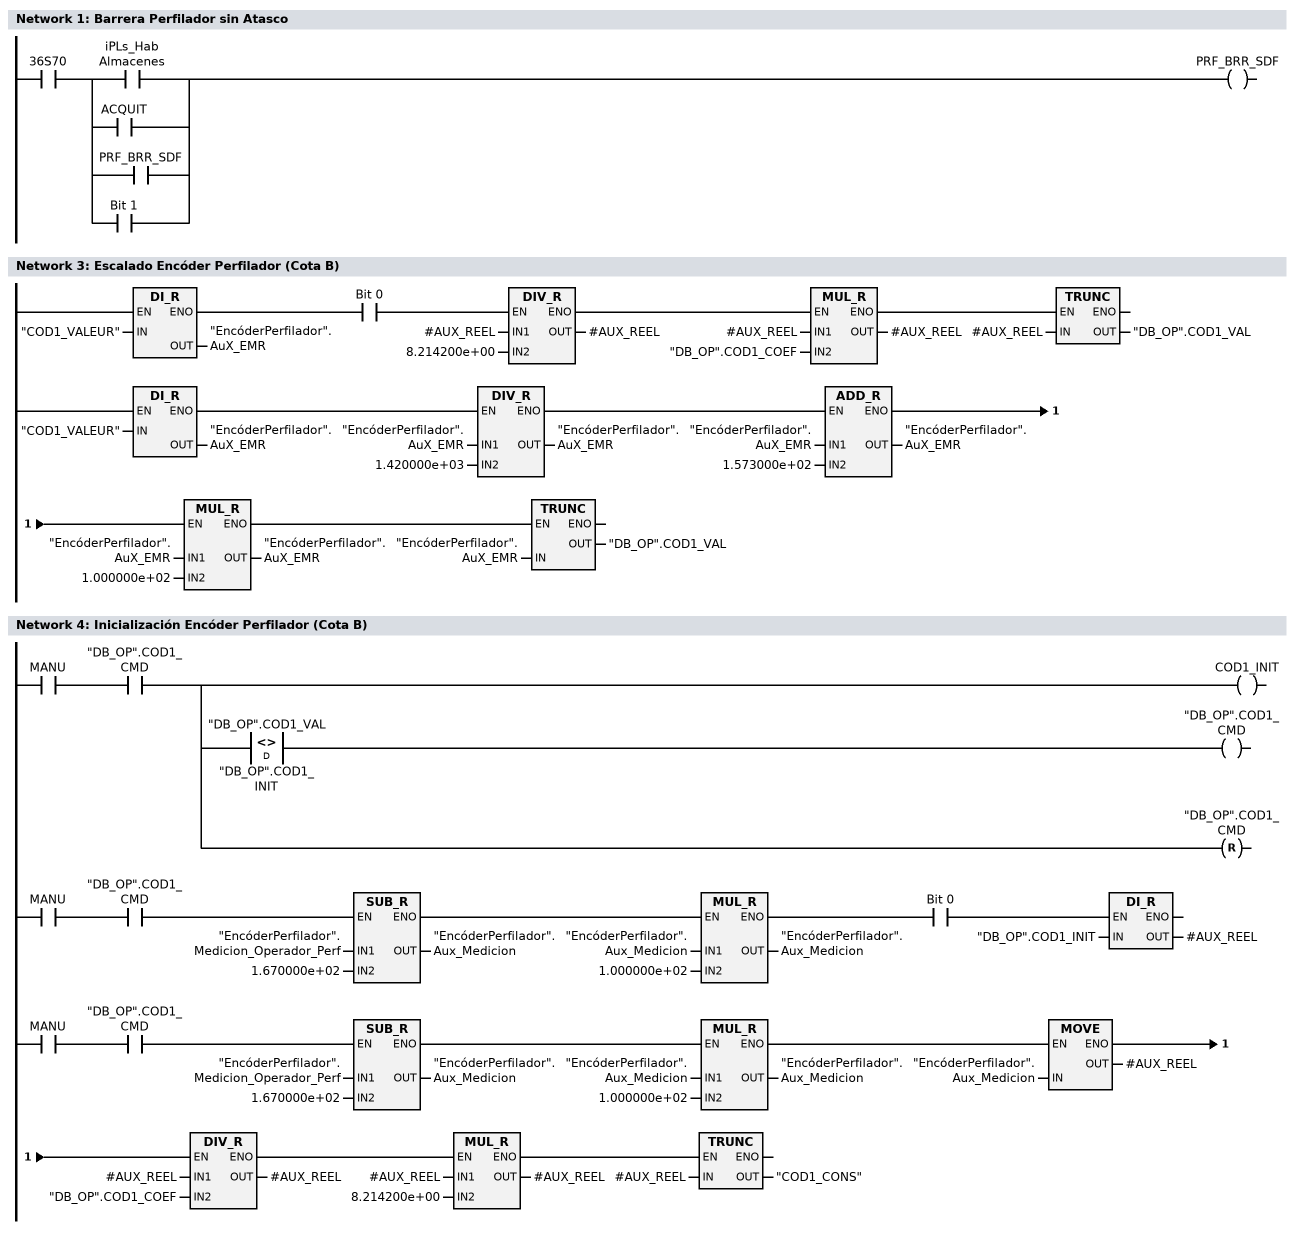
NETWORK
TITLE = Barrera Perfilador sin Atasco
      A     "36S70";
      A(;
      O     "iPLs_HabAlmacenes";
      O     "ACQUIT";
      O     "PRF_BRR_SDF";
      O     "Bit 1";
      );
      =     "PRF_BRR_SDF";
NETWORK
TITLE = Habilitación Infeed Perfiladora (CON/DES1)
      A     "Bit 1";
      A     "KMST";
      =     L 14.0;
      A(;
      A     L 14.0;
      AN    "PRF_SLM_LC";
      AN    "PRF_SLM_LS";
      AN    "PRF_SLM_SH";
      A     "PRF_SLM_BC";
      JNB   _001;
      L     1034;
      T     PQW 24;
      SET;
      SAVE;
      CLR;
_001: A     BR;
      );
      JNB   _002;
      L     1;
      T     PQW 28;
_002: NOP   0;
      A     L 14.0;
      A     "PRF_SLM_LC";
      AN    "PRF_SLM_BC";
      =     L 14.1;
      A(;
      A     L 14.1;
      AN    M 37.7;
      JNB   _003;
      L     1035;
      T     PQW 24;
      SET;
      SAVE;
      CLR;
_003: A     BR;
      );
      JNB   _004;
      L     1;
      T     PQW 28;
_004: NOP   0;
      A(;
      A     L 14.1;
      A     M 37.7;
      JNB   _005;
      L     0;
      T     PQW 24;
      SET;
      SAVE;
      CLR;
_005: A     BR;
      );
      JNB   _006;
      L     1;
      T     PQW 28;
_006: NOP   0;
NETWORK
TITLE = Escalado Encóder Perfilador (Cota B)
      L     "COD1_VALEUR";
      DTR;
      T     "EncóderPerfilador".AuX_EMR;
      SET;
      SAVE;
      CLR;
      A     BR;
      =     L 14.0;
      A(;
      A(;
      A     L 14.0;
      A     "Bit 0";
      JNB   _007;
      L     #AUX_REEL;
      L     8.214200e+00;
      /R;
      T     #AUX_REEL;
      AN    OV;
      SAVE;
      CLR;
_007: A     BR;
      );
      JNB   _008;
      L     #AUX_REEL;
      L     "DB_OP".COD1_COEF;
      *R;
      T     #AUX_REEL;
      AN    OV;
      SAVE;
      CLR;
_008: A     BR;
      );
      JNB   _009;
      L     #AUX_REEL;
      TRUNC;
      T     "DB_OP".COD1_VAL;
_009: NOP   0;
      A(;
      A(;
      A(;
      A     L 14.0;
      JNB   _00a;
      L     "EncóderPerfilador".AuX_EMR;
      L     1.420000e+03;
      /R;
      T     "EncóderPerfilador".AuX_EMR;
      AN    OV;
      SAVE;
      CLR;
_00a: A     BR;
      );
      JNB   _00b;
      L     "EncóderPerfilador".AuX_EMR;
      L     1.573000e+02;
      +R;
      T     "EncóderPerfilador".AuX_EMR;
      AN    OV;
      SAVE;
      CLR;
_00b: A     BR;
      );
      JNB   _00c;
      L     "EncóderPerfilador".AuX_EMR;
      L     1.000000e+02;
      *R;
      T     "EncóderPerfilador".AuX_EMR;
      AN    OV;
      SAVE;
      CLR;
_00c: A     BR;
      );
      JNB   _00d;
      L     "EncóderPerfilador".AuX_EMR;
      TRUNC;
      T     "DB_OP".COD1_VAL;
_00d: NOP   0;
NETWORK
TITLE = Inicialización Encóder Perfilador (Cota B)
      A     "MANU";
      A     "DB_OP".COD1_CMD;
      =     L 14.0;
      A(;
      A     L 14.0;
      JNB   _00e;
      L     "EncóderPerfilador".Medicion_Operador_Perf;
      L     1.670000e+02;
      -R;
      T     "EncóderPerfilador".Aux_Medicion;
      AN    OV;
      SAVE;
      CLR;
_00e: A     BR;
      );
      JNB   _00f;
      L     "EncóderPerfilador".Aux_Medicion;
      L     1.000000e+02;
      *R;
      T     "EncóderPerfilador".Aux_Medicion;
      AN    OV;
      SAVE;
      CLR;
_00f: A     BR;
      =     L 14.1;
      A     L 14.1;
      A     "Bit 0";
      JNB   _010;
      L     "DB_OP".COD1_INIT;
      DTR;
      T     #AUX_REEL;
_010: NOP   0;
      A(;
      A(;
      A(;
      A     L 14.1;
      JNB   _011;
      L     "EncóderPerfilador".Aux_Medicion;
      T     #AUX_REEL;
      SET;
      SAVE;
      CLR;
_011: A     BR;
      );
      JNB   _012;
      L     #AUX_REEL;
      L     "DB_OP".COD1_COEF;
      /R;
      T     #AUX_REEL;
      AN    OV;
      SAVE;
      CLR;
_012: A     BR;
      );
      JNB   _013;
      L     #AUX_REEL;
      L     8.214200e+00;
      *R;
      T     #AUX_REEL;
      AN    OV;
      SAVE;
      CLR;
_013: A     BR;
      );
      JNB   _014;
      L     #AUX_REEL;
      TRUNC;
      T     "COD1_CONS";
_014: NOP   0;
      A     L 14.0;
      BLD   102;
      =     "COD1_INIT";
      A     L 14.0;
      A(;
      L     "DB_OP".COD1_VAL;
      L     "DB_OP".COD1_INIT;
      <>D;
      );
      =     "DB_OP".COD1_CMD;
      A     L 14.0;
      BLD   102;
      R     "DB_OP".COD1_CMD;
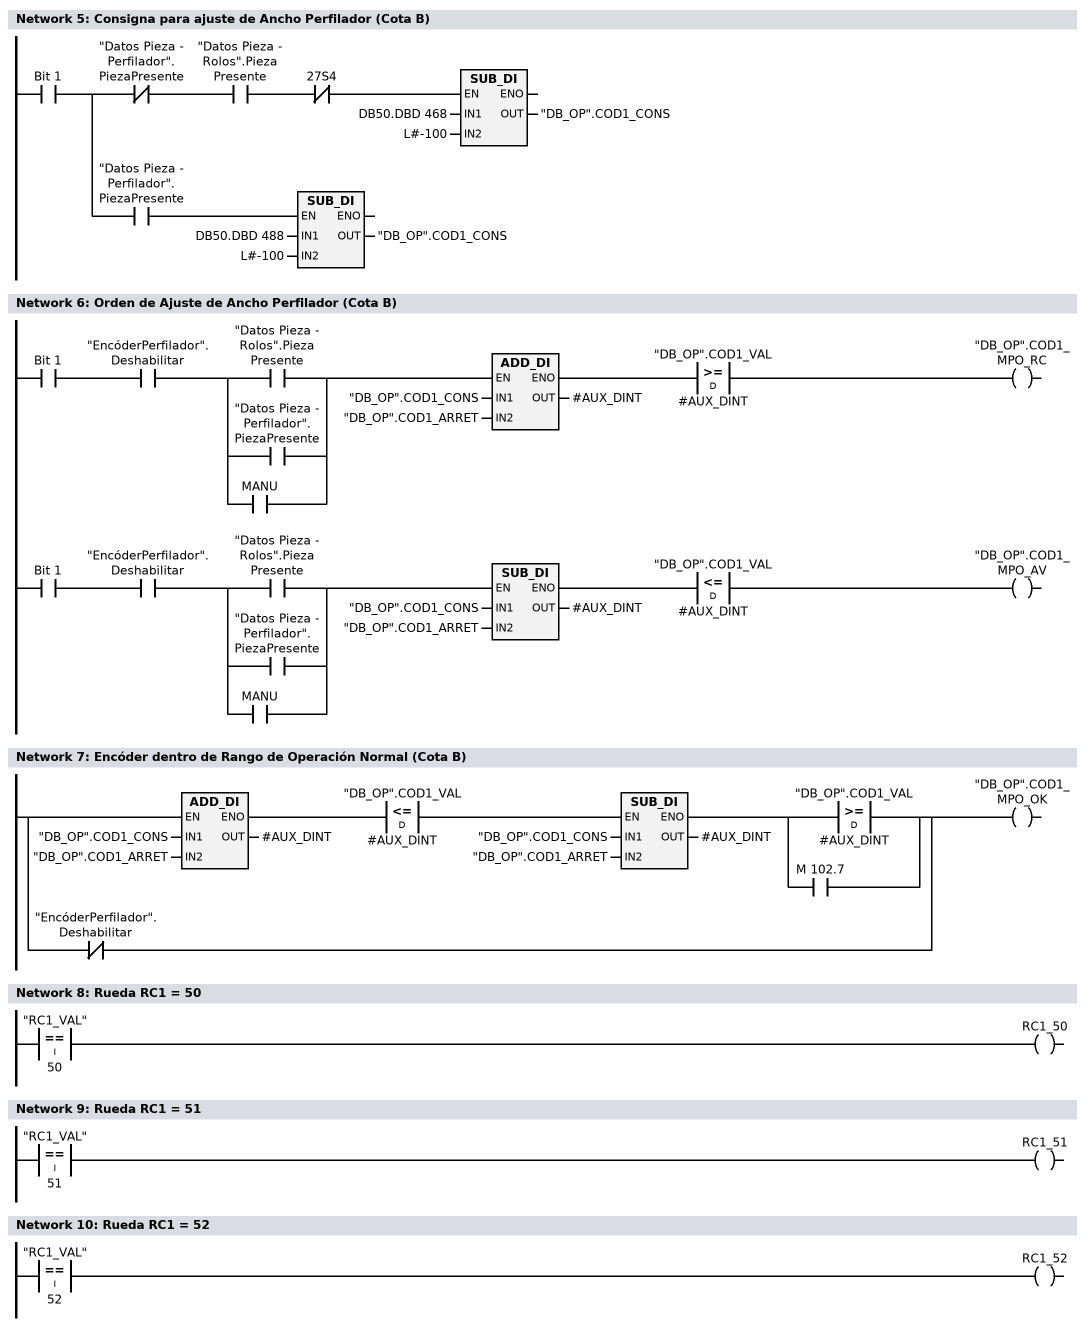
NETWORK
TITLE = Consigna para ajuste de Ancho Perfilador (Cota B)
      A     "Bit 1";
      =     L 14.0;
      A     L 14.0;
      AN    "Datos Pieza - Perfilador".PiezaPresente;
      A     "Datos Pieza - Rolos".PiezaPresente;
      AN    "27S4";
      JNB   _015;
      L     DB50.DBD 468;
      L     L#-100;
      -D;
      T     "DB_OP".COD1_CONS;
_015: NOP   0;
      A     L 14.0;
      A     "Datos Pieza - Perfilador".PiezaPresente;
      JNB   _016;
      L     DB50.DBD 488;
      L     L#-100;
      -D;
      T     "DB_OP".COD1_CONS;
_016: NOP   0;
NETWORK
TITLE = Orden de Ajuste de Ancho Perfilador (Cota B)
      A     "Bit 1";
      A     "EncóderPerfilador".Deshabilitar;
      A(;
      O     "Datos Pieza - Rolos".PiezaPresente;
      O     "Datos Pieza - Perfilador".PiezaPresente;
      O     "MANU";
      );
      =     L 14.0;
      A(;
      A     L 14.0;
      JNB   _017;
      L     "DB_OP".COD1_CONS;
      L     "DB_OP".COD1_ARRET;
      +D;
      T     #AUX_DINT;
      AN    OV;
      SAVE;
      CLR;
_017: A     BR;
      );
      A(;
      L     "DB_OP".COD1_VAL;
      L     #AUX_DINT;
      >=D;
      );
      =     "DB_OP".COD1_MPO_RC;
      A(;
      A     L 14.0;
      JNB   _018;
      L     "DB_OP".COD1_CONS;
      L     "DB_OP".COD1_ARRET;
      -D;
      T     #AUX_DINT;
      AN    OV;
      SAVE;
      CLR;
_018: A     BR;
      );
      A(;
      L     "DB_OP".COD1_VAL;
      L     #AUX_DINT;
      <=D;
      );
      =     "DB_OP".COD1_MPO_AV;
NETWORK
TITLE = Encóder dentro de Rango de Operación Normal (Cota B)
      A(;
      A(;
      L     "DB_OP".COD1_CONS;
      L     "DB_OP".COD1_ARRET;
      +D;
      T     #AUX_DINT;
      AN    OV;
      SAVE;
      CLR;
      A     BR;
      );
      A(;
      L     "DB_OP".COD1_VAL;
      L     #AUX_DINT;
      <=D;
      );
      JNB   _019;
      L     "DB_OP".COD1_CONS;
      L     "DB_OP".COD1_ARRET;
      -D;
      T     #AUX_DINT;
      AN    OV;
      SAVE;
      CLR;
_019: A     BR;
      );
      A(;
      O(;
      L     "DB_OP".COD1_VAL;
      L     #AUX_DINT;
      >=D;
      );
      O     M 102.7;
      );
      ON    "EncóderPerfilador".Deshabilitar;
      =     "DB_OP".COD1_MPO_OK;
NETWORK
TITLE = Rueda RC1 = 50
      L     "RC1_VAL";
      L     50;
      ==I;
      =     "RC1_50";
NETWORK
TITLE = Rueda RC1 = 51
      L     "RC1_VAL";
      L     51;
      ==I;
      =     "RC1_51";
NETWORK
TITLE = Rueda RC1 = 52
      L     "RC1_VAL";
      L     52;
      ==I;
      =     "RC1_52";
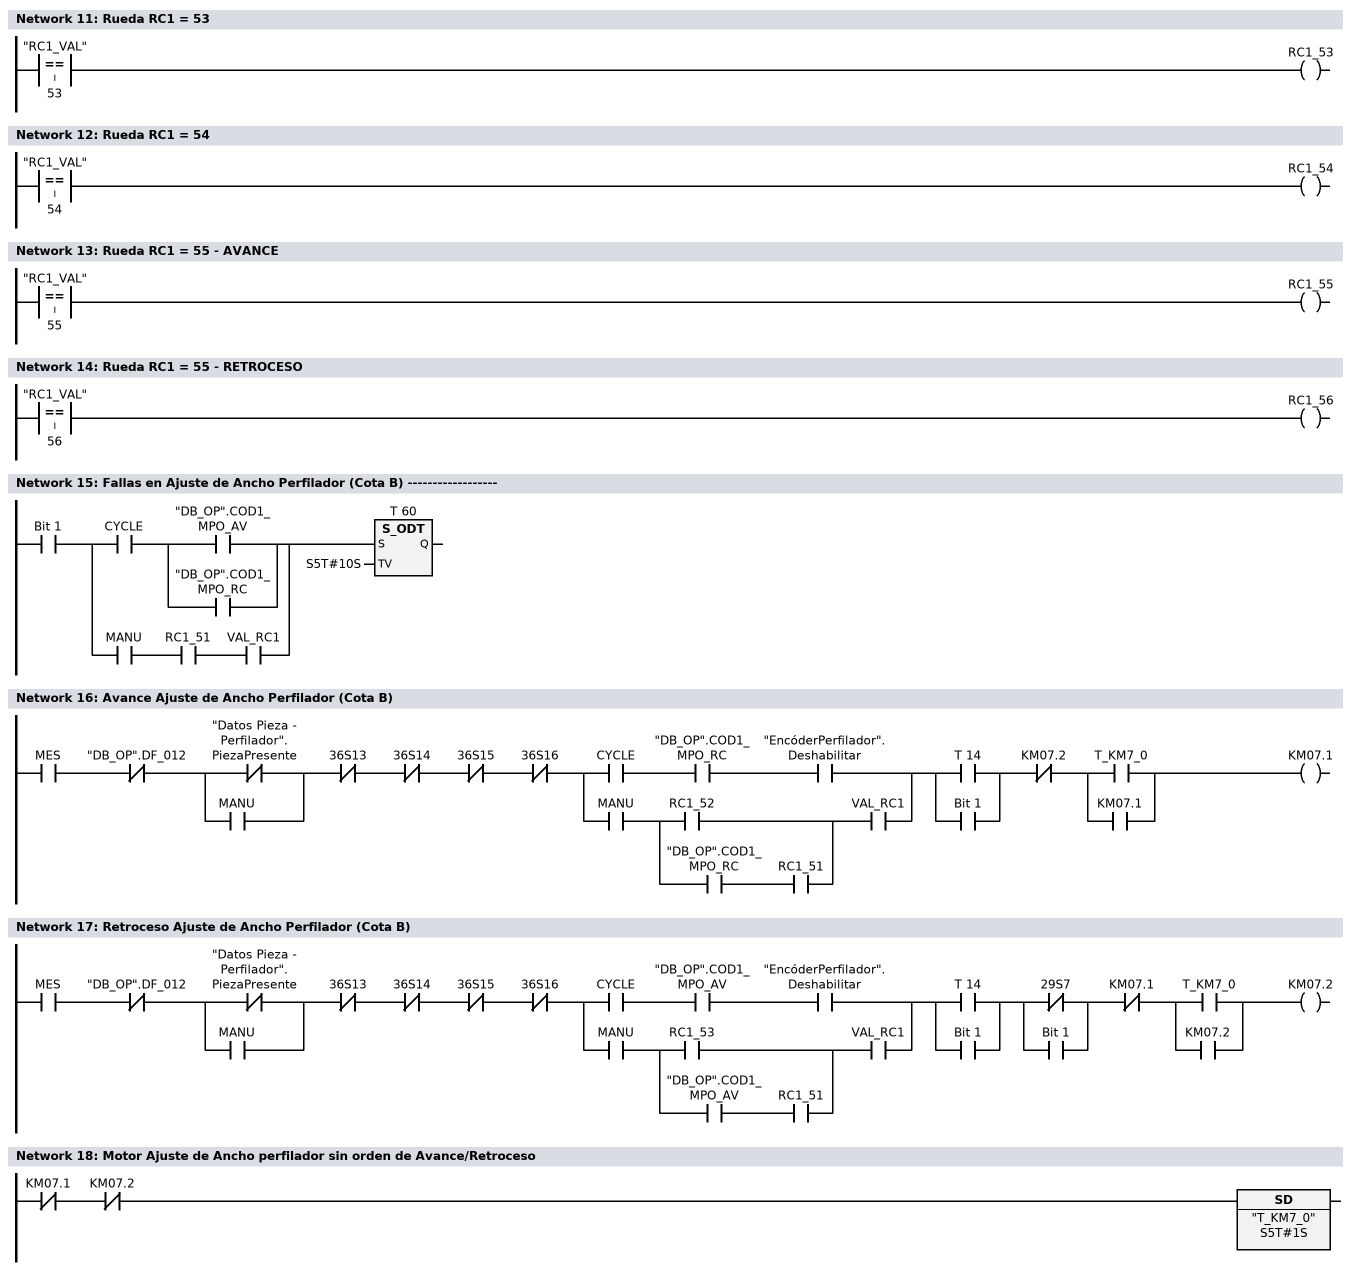
NETWORK
TITLE = Rueda RC1 = 53
      L     "RC1_VAL";
      L     53;
      ==I;
      =     "RC1_53";
NETWORK
TITLE = Rueda RC1 = 54
      L     "RC1_VAL";
      L     54;
      ==I;
      =     "RC1_54";
NETWORK
TITLE = Rueda RC1 = 55 - AVANCE
      L     "RC1_VAL";
      L     55;
      ==I;
      =     "RC1_55";
NETWORK
TITLE = Rueda RC1 = 55 - RETROCESO
      L     "RC1_VAL";
      L     56;
      ==I;
      =     "RC1_56";
NETWORK
TITLE = Fallas en Ajuste de Ancho Perfilador (Cota B) ------------------
      A     "Bit 1";
      A(;
      A     "CYCLE";
      A(;
      O     "DB_OP".COD1_MPO_AV;
      O     "DB_OP".COD1_MPO_RC;
      );
      O;
      A     "MANU";
      A     "RC1_51";
      A     "VAL_RC1";
      );
      L     S5T#10S;
      SD    T 60;
      NOP   0;
      NOP   0;
      NOP   0;
      NOP   0;
NETWORK
TITLE = Avance Ajuste de Ancho Perfilador (Cota B)
      A     "MES";
      AN    "DB_OP".DF_012;
      A(;
      ON    "Datos Pieza - Perfilador".PiezaPresente;
      O     "MANU";
      );
      AN    "36S13";
      AN    "36S14";
      AN    "36S15";
      AN    "36S16";
      A(;
      A     "CYCLE";
      A     "DB_OP".COD1_MPO_RC;
      A     "EncóderPerfilador".Deshabilitar;
      O;
      A     "MANU";
      A(;
      O     "RC1_52";
      O;
      A     "DB_OP".COD1_MPO_RC;
      A     "RC1_51";
      );
      A     "VAL_RC1";
      );
      A(;
      O     T 14;
      O     "Bit 1";
      );
      AN    "KM07.2";
      A(;
      O     "T_KM7_0";
      O     "KM07.1";
      );
      =     "KM07.1";
NETWORK
TITLE = Retroceso Ajuste de Ancho Perfilador (Cota B)
      A     "MES";
      AN    "DB_OP".DF_012;
      A(;
      ON    "Datos Pieza - Perfilador".PiezaPresente;
      O     "MANU";
      );
      AN    "36S13";
      AN    "36S14";
      AN    "36S15";
      AN    "36S16";
      A(;
      A     "CYCLE";
      A     "DB_OP".COD1_MPO_AV;
      A     "EncóderPerfilador".Deshabilitar;
      O;
      A     "MANU";
      A(;
      O     "RC1_53";
      O;
      A     "DB_OP".COD1_MPO_AV;
      A     "RC1_51";
      );
      A     "VAL_RC1";
      );
      A(;
      O     T 14;
      O     "Bit 1";
      );
      A(;
      ON    "29S7";
      O     "Bit 1";
      );
      AN    "KM07.1";
      A(;
      O     "T_KM7_0";
      O     "KM07.2";
      );
      =     "KM07.2";
NETWORK
TITLE = Motor Ajuste de Ancho perfilador sin orden de Avance/Retroceso
      AN    "KM07.1";
      AN    "KM07.2";
      L     S5T#1S;
      SD    "T_KM7_0";
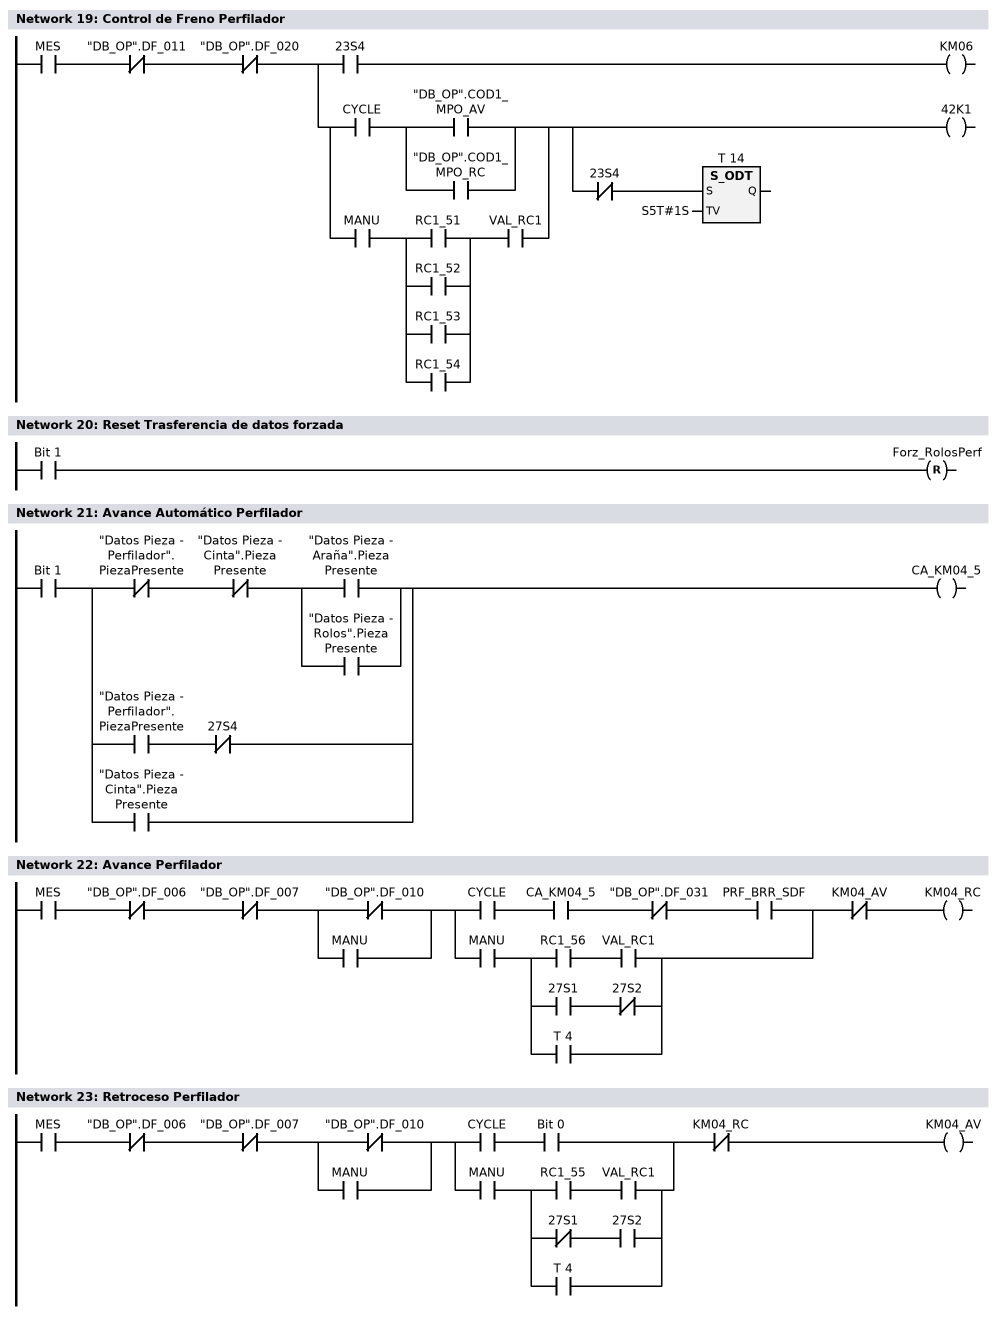
NETWORK
TITLE = Control de Freno Perfilador
      A     "MES";
      AN    "DB_OP".DF_011;
      AN    "DB_OP".DF_020;
      =     L 14.0;
      A     L 14.0;
      A     "23S4";
      =     "KM06";
      A     L 14.0;
      A(;
      A     "CYCLE";
      A(;
      O     "DB_OP".COD1_MPO_AV;
      O     "DB_OP".COD1_MPO_RC;
      );
      O;
      A     "MANU";
      A(;
      O     "RC1_51";
      O     "RC1_52";
      O     "RC1_53";
      O     "RC1_54";
      );
      A     "VAL_RC1";
      );
      =     L 14.1;
      A     L 14.1;
      BLD   102;
      =     "42K1";
      A     L 14.1;
      AN    "23S4";
      L     S5T#1S;
      SD    T 14;
      NOP   0;
      NOP   0;
      NOP   0;
      NOP   0;
NETWORK
TITLE = Reset Trasferencia de datos forzada
      A     "Bit 1";
      R     "Forz_RolosPerf";
NETWORK
TITLE = Avance Automático Perfilador
      A     "Bit 1";
      A(;
      AN    "Datos Pieza - Perfilador".PiezaPresente;
      AN    "Datos Pieza - Cinta".PiezaPresente;
      A(;
      O     "Datos Pieza - Araña".PiezaPresente;
      O     "Datos Pieza - Rolos".PiezaPresente;
      );
      O;
      A     "Datos Pieza - Perfilador".PiezaPresente;
      AN    "27S4";
      O     "Datos Pieza - Cinta".PiezaPresente;
      );
      =     "CA_KM04_5";
NETWORK
TITLE = Avance Perfilador
      A     "MES";
      AN    "DB_OP".DF_006;
      AN    "DB_OP".DF_007;
      A(;
      ON    "DB_OP".DF_010;
      O     "MANU";
      );
      A(;
      A     "CYCLE";
      A     "CA_KM04_5";
      AN    "DB_OP".DF_031;
      A     "PRF_BRR_SDF";
      O;
      A     "MANU";
      A(;
      A     "RC1_56";
      A     "VAL_RC1";
      O;
      A     "27S1";
      AN    "27S2";
      O     T 4;
      );
      );
      AN    "KM04_AV";
      =     "KM04_RC";
NETWORK
TITLE = Retroceso Perfilador
      A     "MES";
      AN    "DB_OP".DF_006;
      AN    "DB_OP".DF_007;
      A(;
      ON    "DB_OP".DF_010;
      O     "MANU";
      );
      A(;
      A     "CYCLE";
      A     "Bit 0";
      O;
      A     "MANU";
      A(;
      A     "RC1_55";
      A     "VAL_RC1";
      O;
      AN    "27S1";
      A     "27S2";
      O     T 4;
      );
      );
      AN    "KM04_RC";
      =     "KM04_AV";
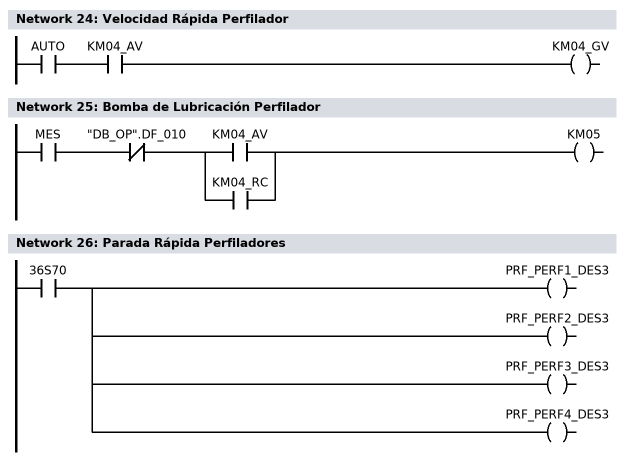
NETWORK
TITLE = Velocidad Rápida Perfilador
      A     "AUTO";
      A     "KM04_AV";
      =     "KM04_GV";
NETWORK
TITLE = Bomba de Lubricación Perfilador
      A     "MES";
      AN    "DB_OP".DF_010;
      A(;
      O     "KM04_AV";
      O     "KM04_RC";
      );
      =     "KM05";
NETWORK
TITLE = Parada Rápida Perfiladores
      A     "36S70";
      =     "PRF_PERF1_DES3";
      =     "PRF_PERF2_DES3";
      =     "PRF_PERF3_DES3";
      =     "PRF_PERF4_DES3";
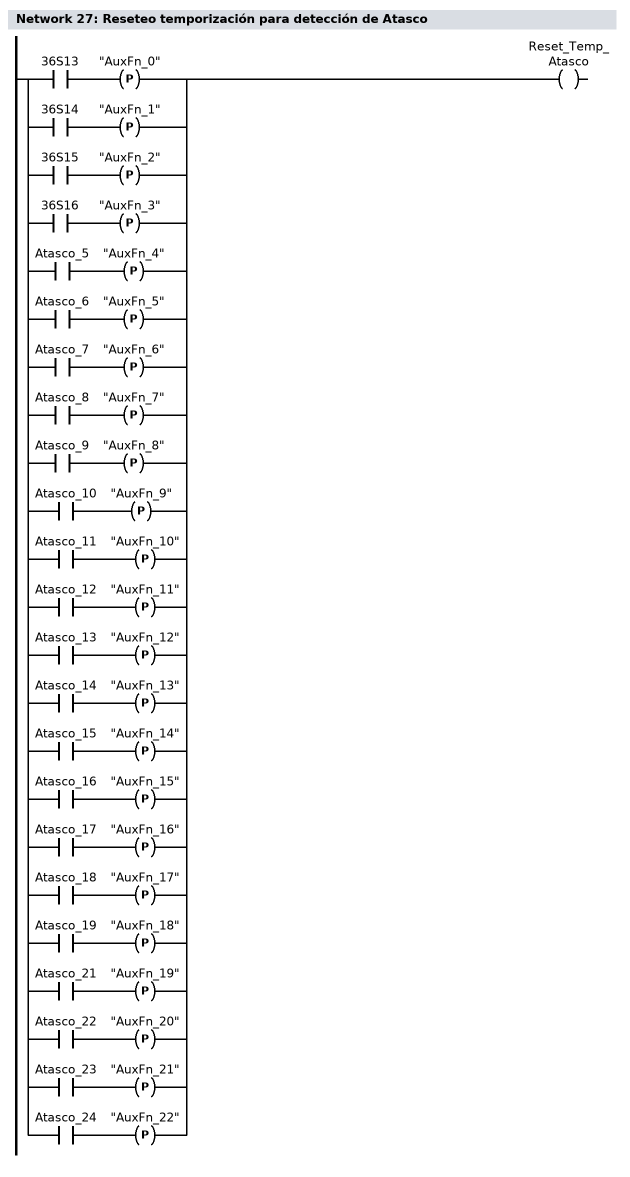
NETWORK
TITLE = Reseteo temporización para detección de Atasco
      A     "36S13";
      FP    "AuxFn_0";
      O(;
      A     "36S14";
      FP    "AuxFn_1";
      );
      O(;
      A     "36S15";
      FP    "AuxFn_2";
      );
      O(;
      A     "36S16";
      FP    "AuxFn_3";
      );
      O(;
      A     "Atasco_5";
      FP    "AuxFn_4";
      );
      O(;
      A     "Atasco_6";
      FP    "AuxFn_5";
      );
      O(;
      A     "Atasco_7";
      FP    "AuxFn_6";
      );
      O(;
      A     "Atasco_8";
      FP    "AuxFn_7";
      );
      O(;
      A     "Atasco_9";
      FP    "AuxFn_8";
      );
      O(;
      A     "Atasco_10";
      FP    "AuxFn_9";
      );
      O(;
      A     "Atasco_11";
      FP    "AuxFn_10";
      );
      O(;
      A     "Atasco_12";
      FP    "AuxFn_11";
      );
      O(;
      A     "Atasco_13";
      FP    "AuxFn_12";
      );
      O(;
      A     "Atasco_14";
      FP    "AuxFn_13";
      );
      O(;
      A     "Atasco_15";
      FP    "AuxFn_14";
      );
      O(;
      A     "Atasco_16";
      FP    "AuxFn_15";
      );
      O(;
      A     "Atasco_17";
      FP    "AuxFn_16";
      );
      O(;
      A     "Atasco_18";
      FP    "AuxFn_17";
      );
      O(;
      A     "Atasco_19";
      FP    "AuxFn_18";
      );
      O(;
      A     "Atasco_21";
      FP    "AuxFn_19";
      );
      O(;
      A     "Atasco_22";
      FP    "AuxFn_20";
      );
      O(;
      A     "Atasco_23";
      FP    "AuxFn_21";
      );
      O(;
      A     "Atasco_24";
      FP    "AuxFn_22";
      );
      =     "Reset_Temp_Atasco";
END_FUNCTION

FUNCTION "Transportes" : VOID	// FC 11
TITLE = Transportes
VERSION : 0.1
VAR_TEMP
  SECU : BOOL ;	//Seguridades
  SEL_MANU : BOOL ;	//Modo Manual
  NMVT : INT ;	//Numero Mouvement
  Vitesse : INT ;	//Consigna Velocidad
END_VAR
BEGIN
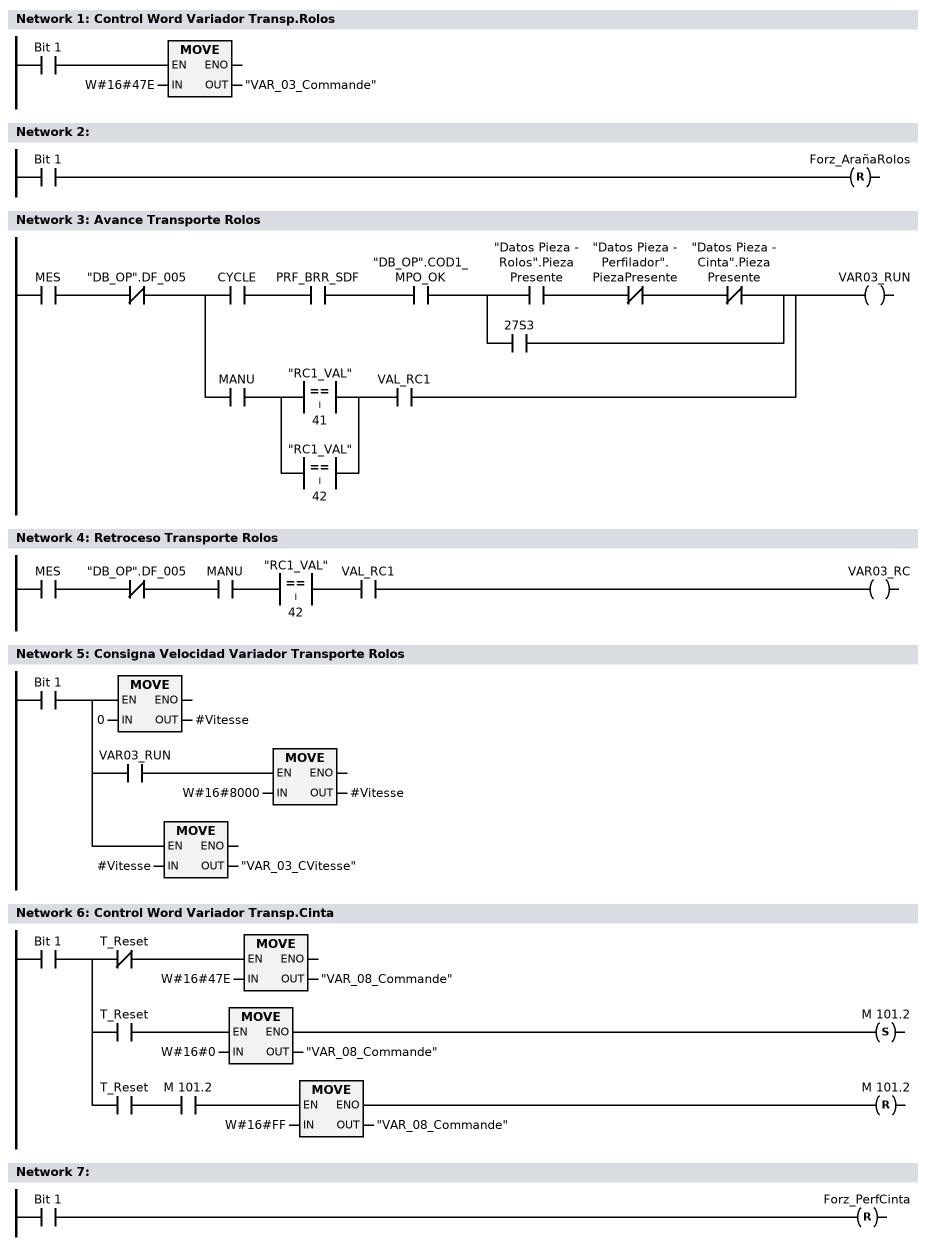
NETWORK
TITLE = Control Word Variador Transp.Rolos
      A     "Bit 1";
      JNB   _001;
      L     W#16#47E;
      T     "VAR_03_Commande";
_001: NOP   0;
NETWORK
TITLE =
      A     "Bit 1";
      R     "Forz_ArañaRolos";
NETWORK
TITLE = Avance Transporte Rolos
      A     "MES";
      AN    "DB_OP".DF_005;
      A(;
      A     "CYCLE";
      A     "PRF_BRR_SDF";
      A     "DB_OP".COD1_MPO_OK;
      A(;
      A     "Datos Pieza - Rolos".PiezaPresente;
      AN    "Datos Pieza - Perfilador".PiezaPresente;
      AN    "Datos Pieza - Cinta".PiezaPresente;
      O     "27S3";
      );
      O;
      A     "MANU";
      A(;
      O(;
      L     "RC1_VAL";
      L     41;
      ==I;
      );
      O(;
      L     "RC1_VAL";
      L     42;
      ==I;
      );
      );
      A     "VAL_RC1";
      );
      =     "VAR03_RUN";
NETWORK
TITLE = Retroceso Transporte Rolos
      A     "MES";
      AN    "DB_OP".DF_005;
      A     "MANU";
      A(;
      L     "RC1_VAL";
      L     42;
      ==I;
      );
      A     "VAL_RC1";
      =     "VAR03_RC";
NETWORK
TITLE = Consigna Velocidad Variador Transporte Rolos
      A     "Bit 1";
      =     L 6.0;
      A     L 6.0;
      JNB   _002;
      L     0;
      T     #Vitesse;
_002: NOP   0;
      A     L 6.0;
      A     "VAR03_RUN";
      JNB   _003;
      L     W#16#8000;
      T     #Vitesse;
_003: NOP   0;
      A     L 6.0;
      JNB   _004;
      L     #Vitesse;
      T     "VAR_03_CVitesse";
_004: NOP   0;
NETWORK
TITLE = Control Word Variador Transp.Cinta 
      A     "Bit 1";
      =     L 6.0;
      A     L 6.0;
      AN    "T_Reset";
      JNB   _005;
      L     W#16#47E;
      T     "VAR_08_Commande";
_005: NOP   0;
      A     L 6.0;
      A     "T_Reset";
      JNB   _006;
      L     W#16#0;
      T     "VAR_08_Commande";
      SET;
      SAVE;
      CLR;
_006: A     BR;
      S     M 101.2;
      A     L 6.0;
      A     "T_Reset";
      A     M 101.2;
      JNB   _007;
      L     W#16#FF;
      T     "VAR_08_Commande";
      SET;
      SAVE;
      CLR;
_007: A     BR;
      R     M 101.2;
NETWORK
TITLE =
      A     "Bit 1";
      R     "Forz_PerfCinta";
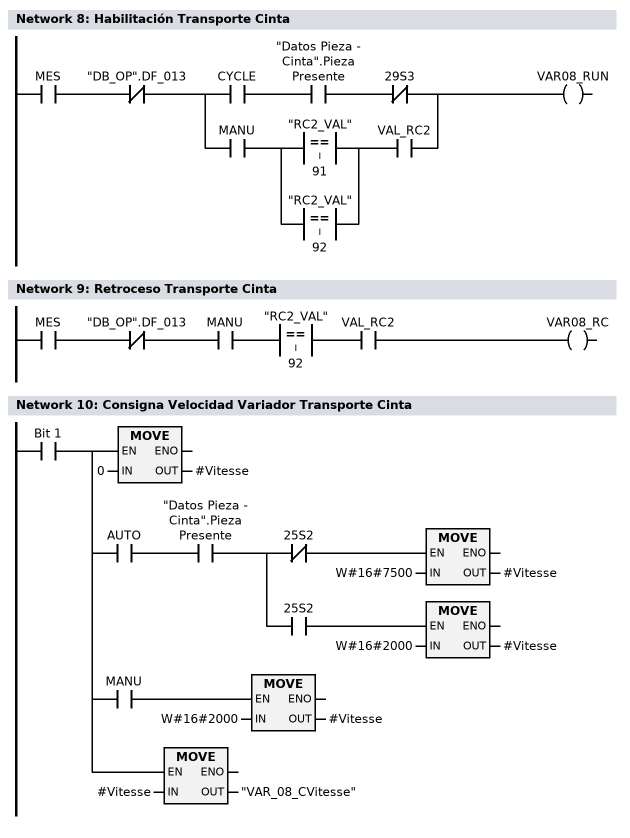
NETWORK
TITLE = Habilitación Transporte Cinta
      A     "MES";
      AN    "DB_OP".DF_013;
      A(;
      A     "CYCLE";
      A     "Datos Pieza - Cinta".PiezaPresente;
      AN    "29S3";
      O;
      A     "MANU";
      A(;
      O(;
      L     "RC2_VAL";
      L     91;
      ==I;
      );
      O(;
      L     "RC2_VAL";
      L     92;
      ==I;
      );
      );
      A     "VAL_RC2";
      );
      =     "VAR08_RUN";
NETWORK
TITLE = Retroceso Transporte Cinta
      A     "MES";
      AN    "DB_OP".DF_013;
      A     "MANU";
      A(;
      L     "RC2_VAL";
      L     92;
      ==I;
      );
      A     "VAL_RC2";
      =     "VAR08_RC";
NETWORK
TITLE = Consigna Velocidad Variador Transporte Cinta
      A     "Bit 1";
      =     L 6.0;
      A     L 6.0;
      JNB   _008;
      L     0;
      T     #Vitesse;
_008: NOP   0;
      A     L 6.0;
      A     "AUTO";
      A     "Datos Pieza - Cinta".PiezaPresente;
      =     L 6.1;
      A     L 6.1;
      AN    "25S2";
      JNB   _009;
      L     W#16#7500;
      T     #Vitesse;
_009: NOP   0;
      A     L 6.1;
      A     "25S2";
      JNB   _00a;
      L     W#16#2000;
      T     #Vitesse;
_00a: NOP   0;
      A     L 6.0;
      A     "MANU";
      JNB   _00b;
      L     W#16#2000;
      T     #Vitesse;
_00b: NOP   0;
      A     L 6.0;
      JNB   _00c;
      L     #Vitesse;
      T     "VAR_08_CVitesse";
_00c: NOP   0;
END_FUNCTION

FUNCTION "Control de Pinza y Forma" : VOID	// FC 12
TITLE = Control de Pinza y Formador
AUTHOR : EMR
NAME : eProC
VERSION : 0.1
VAR_TEMP
  SECU : BOOL ;	//Sécurité mé
  SEL_MANU : BOOL ;	//Sélection m
  TEMP0 : INT ;	//Numero Mouv
  AUX_REEL : REAL ;
  AUX_DINT : DINT ;
  AUX_ENCODER : REAL ;
  AUX_ENCODER2 : DINT ;
  PI_A : DINT ;
  PI_B : DINT ;
  PI_C : DINT ;
  PI_D : DINT ;
  AUX_POS_F4 : DINT ;
  PI_F1 : DINT ;
  PI_F2 : DINT ;
  PI_F3 : DINT ;
  PI_F4 : DINT ;
  AUX_POS_F1 : DINT ;
  AUX_POS_F2 : DINT ;
  AUX_POS_F3 : DINT ;
  AUX_CHAPA_COMPLETA : DINT ;
  AUX_SALIDA : DINT ;
  AUX_REAL : REAL ;
  AUX_ENTREGA : DINT ;
  AUX_POS_RECEP : BOOL ;	//Pos. Recepción dentro de tolerancia
  AUX_POS_ENT : BOOL ;	//Pos. Entrega dentro de tolerancia
  AUX_POS_E2H2 : BOOL ;	//Pos. E2H2 dentro de tolerancia
  AUX_POS_E2H1 : BOOL ;	//Pos. E2H1 dentro de tolerancia
  AUX_POS_E1H2 : BOOL ;	//Pos. E1H2 dentro de tolerancia
  AUX_POS_E1H1 : BOOL ;	//Pos. E1H1 dentro de tolerancia
END_VAR
BEGIN
NETWORK
TITLE = ------------- HABILITACIÓN SERVOS -----------------
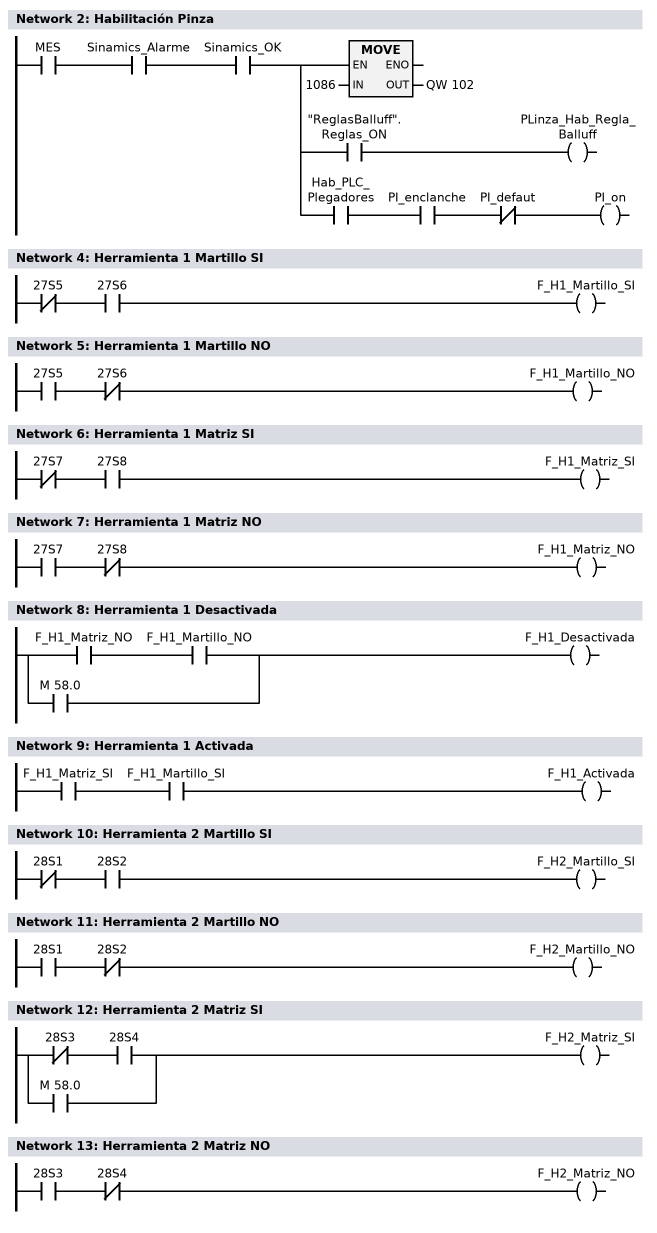
NETWORK
TITLE = Habilitación Pinza
      A     "MES";
      A     "Sinamics_Alarme";
      A     "Sinamics_OK";
      =     L 85.0;
      A     L 85.0;
      JNB   _001;
      L     1086;
      T     QW 102;
_001: NOP   0;
      A     L 85.0;
      A     "ReglasBalluff".Reglas_ON;
      =     "PLinza_Hab_Regla_Balluff";
      A     L 85.0;
      A     "Hab_PLC_Plegadores";
      A     "PI_enclanche";
      AN    "PI_defaut";
      =     "PI_on";
NETWORK
TITLE = ------------- RESUMEN DE SENSORES -----------------
NETWORK
TITLE = Herramienta 1 Martillo SI
      AN    "27S5";
      A     "27S6";
      =     "F_H1_Martillo_SI";
NETWORK
TITLE = Herramienta 1 Martillo NO
      A     "27S5";
      AN    "27S6";
      =     "F_H1_Martillo_NO";
NETWORK
TITLE = Herramienta 1 Matriz SI
      AN    "27S7";
      A     "27S8";
      =     "F_H1_Matriz_SI";
NETWORK
TITLE = Herramienta 1 Matriz NO
      A     "27S7";
      AN    "27S8";
      =     "F_H1_Matriz_NO";
NETWORK
TITLE = Herramienta 1 Desactivada
      A     "F_H1_Matriz_NO";
      A     "F_H1_Martillo_NO";
      O     M 58.0;
      =     "F_H1_Desactivada";
NETWORK
TITLE = Herramienta 1 Activada
      A     "F_H1_Matriz_SI";
      A     "F_H1_Martillo_SI";
      =     "F_H1_Activada";
NETWORK
TITLE = Herramienta 2 Martillo SI
      AN    "28S1";
      A     "28S2";
      =     "F_H2_Martillo_SI";
NETWORK
TITLE = Herramienta 2 Martillo NO
      A     "28S1";
      AN    "28S2";
      =     "F_H2_Martillo_NO";
NETWORK
TITLE = Herramienta 2 Matriz SI
      AN    "28S3";
      A     "28S4";
      O     M 58.0;
      =     "F_H2_Matriz_SI";
NETWORK
TITLE = Herramienta 2 Matriz NO
      A     "28S3";
      AN    "28S4";
      =     "F_H2_Matriz_NO";
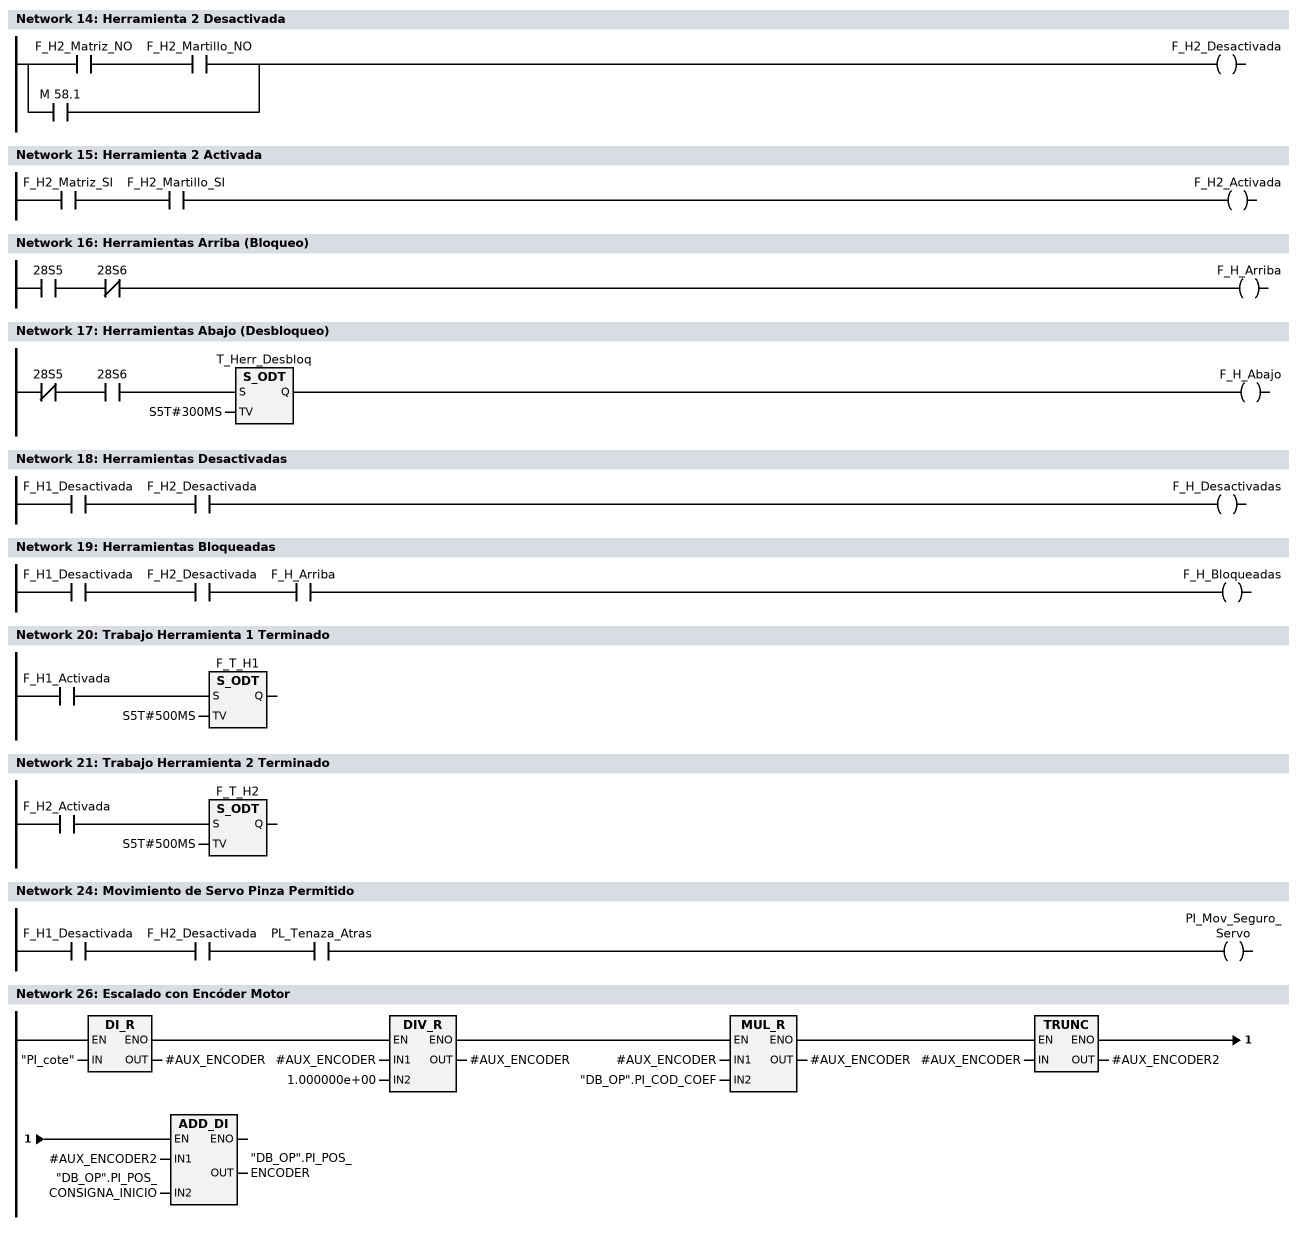
NETWORK
TITLE = Herramienta 2 Desactivada
      A     "F_H2_Matriz_NO";
      A     "F_H2_Martillo_NO";
      O     M 58.1;
      =     "F_H2_Desactivada";
NETWORK
TITLE = Herramienta 2 Activada
      A     "F_H2_Matriz_SI";
      A     "F_H2_Martillo_SI";
      =     "F_H2_Activada";
NETWORK
TITLE = Herramientas Arriba (Bloqueo)
      A     "28S5";
      AN    "28S6";
      =     "F_H_Arriba";
NETWORK
TITLE = Herramientas Abajo (Desbloqueo)
      AN    "28S5";
      A     "28S6";
      L     S5T#300MS;
      SD    "T_Herr_Desbloq";
      NOP   0;
      NOP   0;
      NOP   0;
      A     "T_Herr_Desbloq";
      =     "F_H_Abajo";
NETWORK
TITLE = Herramientas Desactivadas
      A     "F_H1_Desactivada";
      A     "F_H2_Desactivada";
      =     "F_H_Desactivadas";
NETWORK
TITLE = Herramientas Bloqueadas
      A     "F_H1_Desactivada";
      A     "F_H2_Desactivada";
      A     "F_H_Arriba";
      =     "F_H_Bloqueadas";
NETWORK
TITLE = Trabajo Herramienta 1 Terminado
      A     "F_H1_Activada";
      L     S5T#500MS;
      SD    "F_T_H1";
      NOP   0;
      NOP   0;
      NOP   0;
      NOP   0;
NETWORK
TITLE = Trabajo Herramienta 2 Terminado
      A     "F_H2_Activada";
      L     S5T#500MS;
      SD    "F_T_H2";
      NOP   0;
      NOP   0;
      NOP   0;
      NOP   0;
NETWORK
TITLE = Ciclo Formado H1 Finalizado
      A(;
      A     "F_T_H1";
      S     "F_TTH1";
      A(;
      O     "S_F_8";
      O     "S_F_10";
      );
      R     "F_TTH1";
      A     "F_TTH1";
      );
      A     "F_H1_Desactivada";
      =     "F_H1_Ciclo_FIN";
NETWORK
TITLE = Ciclo Formado H2 Finalizado
      A(;
      A     "F_T_H2";
      S     "F_TTH2";
      A(;
      O     "S_F_9";
      O     "S_F_11";
      );
      R     "F_TTH2";
      A     "F_TTH2";
      );
      A     "F_H2_Desactivada";
      =     "F_H2_Ciclo_FIN";
NETWORK
TITLE = Movimiento de Servo Pinza Permitido
      A     "F_H1_Desactivada";
      A     "F_H2_Desactivada";
      A     "PL_Tenaza_Atras";
      =     "PI_Mov_Seguro_Servo";
NETWORK
TITLE = ------------ ESCALADO DE ENCODERS -------------
NETWORK
TITLE = Escalado con Encóder Motor
      A(;
      A(;
      A(;
      A(;
      L     "PI_cote";
      DTR;
      T     #AUX_ENCODER;
      SET;
      SAVE;
      CLR;
      A     BR;
      );
      JNB   _002;
      L     #AUX_ENCODER;
      L     1.000000e+00;
      /R;
      T     #AUX_ENCODER;
      AN    OV;
      SAVE;
      CLR;
_002: A     BR;
      );
      JNB   _003;
      L     #AUX_ENCODER;
      L     "DB_OP".PI_COD_COEF;
      *R;
      T     #AUX_ENCODER;
      AN    OV;
      SAVE;
      CLR;
_003: A     BR;
      );
      JNB   _004;
      L     #AUX_ENCODER;
      TRUNC;
      T     #AUX_ENCODER2;
      AN    OV;
      SAVE;
      CLR;
_004: A     BR;
      );
      JNB   _005;
      L     #AUX_ENCODER2;
      L     "DB_OP".PI_POS_CONSIGNA_INICIO;
      +D;
      T     "DB_OP".PI_POS_ENCODER;
_005: NOP   0;
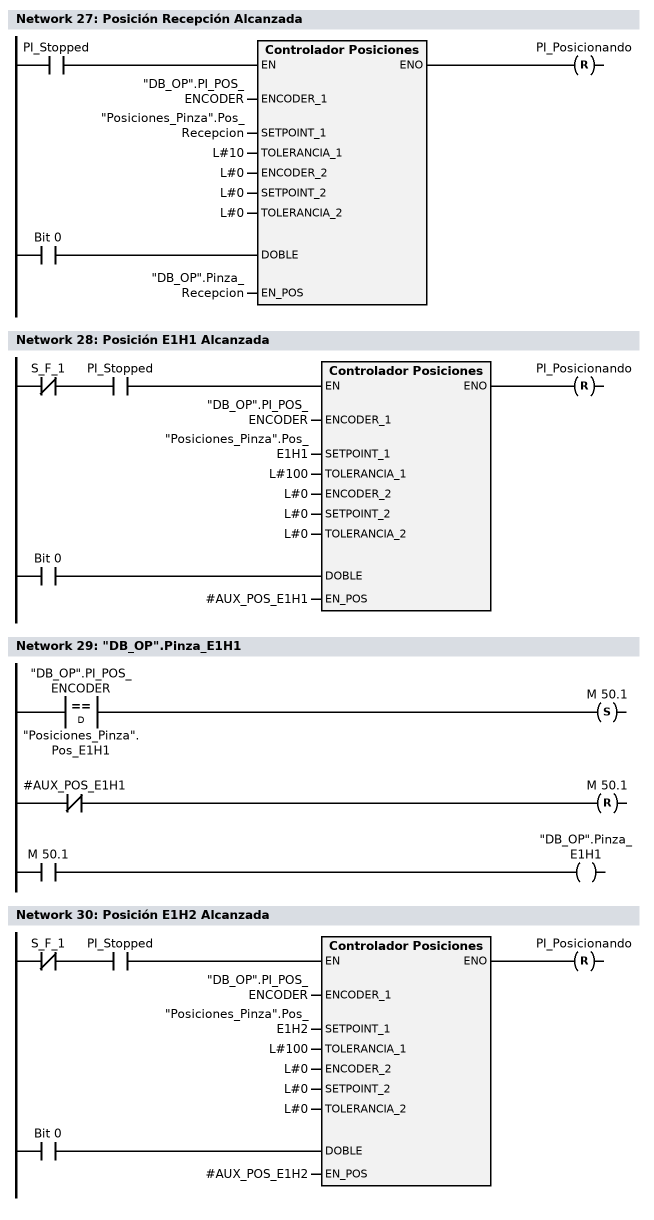
NETWORK
TITLE = Posición Recepción Alcanzada
      A     "Bit 0";
      =     L 85.0;
      BLD   103;
      A     "PI_Stopped";
      JNB   _006;
      CALL  "Controlador Posiciones" (
           ENCODER_1                := "DB_OP".PI_POS_ENCODER,
           SETPOINT_1               := "Posiciones_Pinza".Pos_Recepcion,
           TOLERANCIA_1             := L#10,
           ENCODER_2                := L#0,
           SETPOINT_2               := L#0,
           TOLERANCIA_2             := L#0,
           DOBLE                    := L 85.0,
           EN_POS                   := "DB_OP".Pinza_Recepcion);
_006: A     BR;
      R     "PI_Posicionando";
NETWORK
TITLE = Posición E1H1 Alcanzada
      A     "Bit 0";
      =     L 85.0;
      BLD   103;
      AN    "S_F_1";
      A     "PI_Stopped";
      JNB   _007;
      CALL  "Controlador Posiciones" (
           ENCODER_1                := "DB_OP".PI_POS_ENCODER,
           SETPOINT_1               := "Posiciones_Pinza".Pos_E1H1,
           TOLERANCIA_1             := L#100,
           ENCODER_2                := L#0,
           SETPOINT_2               := L#0,
           TOLERANCIA_2             := L#0,
           DOBLE                    := L 85.0,
           EN_POS                   := #AUX_POS_E1H1);
_007: A     BR;
      R     "PI_Posicionando";
NETWORK
TITLE = "DB_OP".Pinza_E1H1
      A(;
      L     "DB_OP".PI_POS_ENCODER;
      L     "Posiciones_Pinza".Pos_E1H1;
      ==D;
      );
      S     M 50.1;
      AN    #AUX_POS_E1H1;
      R     M 50.1;
      A     M 50.1;
      =     "DB_OP".Pinza_E1H1;
NETWORK
TITLE = Posición E1H2 Alcanzada
      A     "Bit 0";
      =     L 85.0;
      BLD   103;
      AN    "S_F_1";
      A     "PI_Stopped";
      JNB   _008;
      CALL  "Controlador Posiciones" (
           ENCODER_1                := "DB_OP".PI_POS_ENCODER,
           SETPOINT_1               := "Posiciones_Pinza".Pos_E1H2,
           TOLERANCIA_1             := L#100,
           ENCODER_2                := L#0,
           SETPOINT_2               := L#0,
           TOLERANCIA_2             := L#0,
           DOBLE                    := L 85.0,
           EN_POS                   := #AUX_POS_E1H2);
_008: A     BR;
      R     "PI_Posicionando";
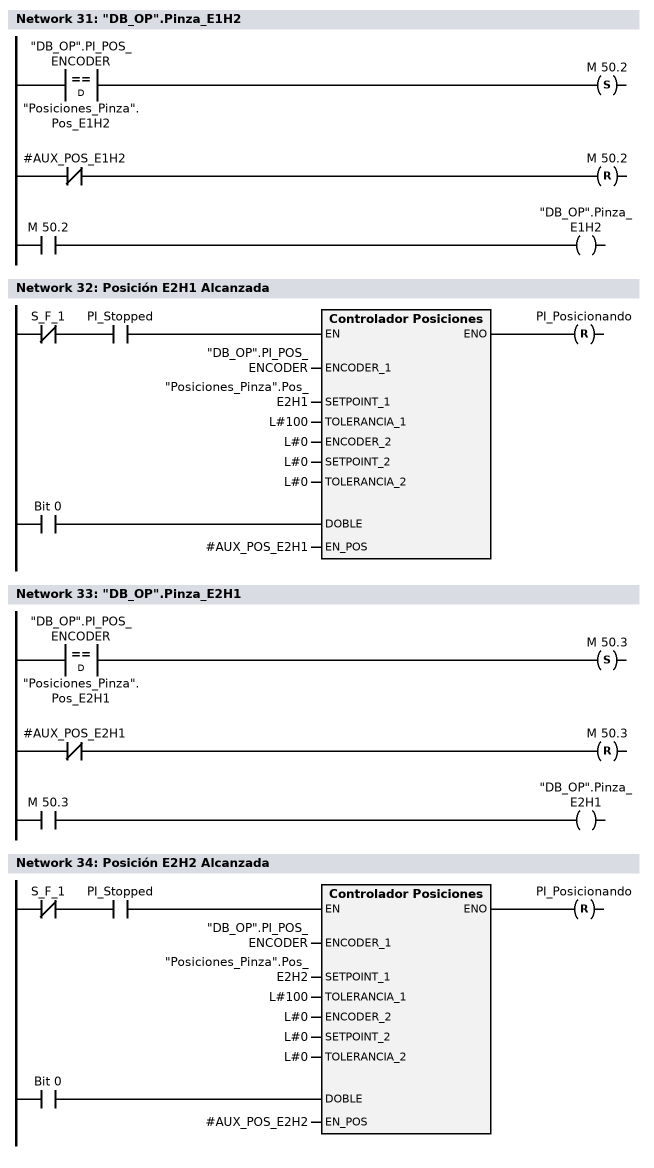
NETWORK
TITLE = "DB_OP".Pinza_E1H2
      A(;
      L     "DB_OP".PI_POS_ENCODER;
      L     "Posiciones_Pinza".Pos_E1H2;
      ==D;
      );
      S     M 50.2;
      AN    #AUX_POS_E1H2;
      R     M 50.2;
      A     M 50.2;
      =     "DB_OP".Pinza_E1H2;
NETWORK
TITLE = Posición E2H1 Alcanzada
      A     "Bit 0";
      =     L 85.0;
      BLD   103;
      AN    "S_F_1";
      A     "PI_Stopped";
      JNB   _009;
      CALL  "Controlador Posiciones" (
           ENCODER_1                := "DB_OP".PI_POS_ENCODER,
           SETPOINT_1               := "Posiciones_Pinza".Pos_E2H1,
           TOLERANCIA_1             := L#100,
           ENCODER_2                := L#0,
           SETPOINT_2               := L#0,
           TOLERANCIA_2             := L#0,
           DOBLE                    := L 85.0,
           EN_POS                   := #AUX_POS_E2H1);
_009: A     BR;
      R     "PI_Posicionando";
NETWORK
TITLE = "DB_OP".Pinza_E2H1
      A(;
      L     "DB_OP".PI_POS_ENCODER;
      L     "Posiciones_Pinza".Pos_E2H1;
      ==D;
      );
      S     M 50.3;
      AN    #AUX_POS_E2H1;
      R     M 50.3;
      A     M 50.3;
      =     "DB_OP".Pinza_E2H1;
NETWORK
TITLE = Posición E2H2 Alcanzada
      A     "Bit 0";
      =     L 85.0;
      BLD   103;
      AN    "S_F_1";
      A     "PI_Stopped";
      JNB   _00a;
      CALL  "Controlador Posiciones" (
           ENCODER_1                := "DB_OP".PI_POS_ENCODER,
           SETPOINT_1               := "Posiciones_Pinza".Pos_E2H2,
           TOLERANCIA_1             := L#100,
           ENCODER_2                := L#0,
           SETPOINT_2               := L#0,
           TOLERANCIA_2             := L#0,
           DOBLE                    := L 85.0,
           EN_POS                   := #AUX_POS_E2H2);
_00a: A     BR;
      R     "PI_Posicionando";
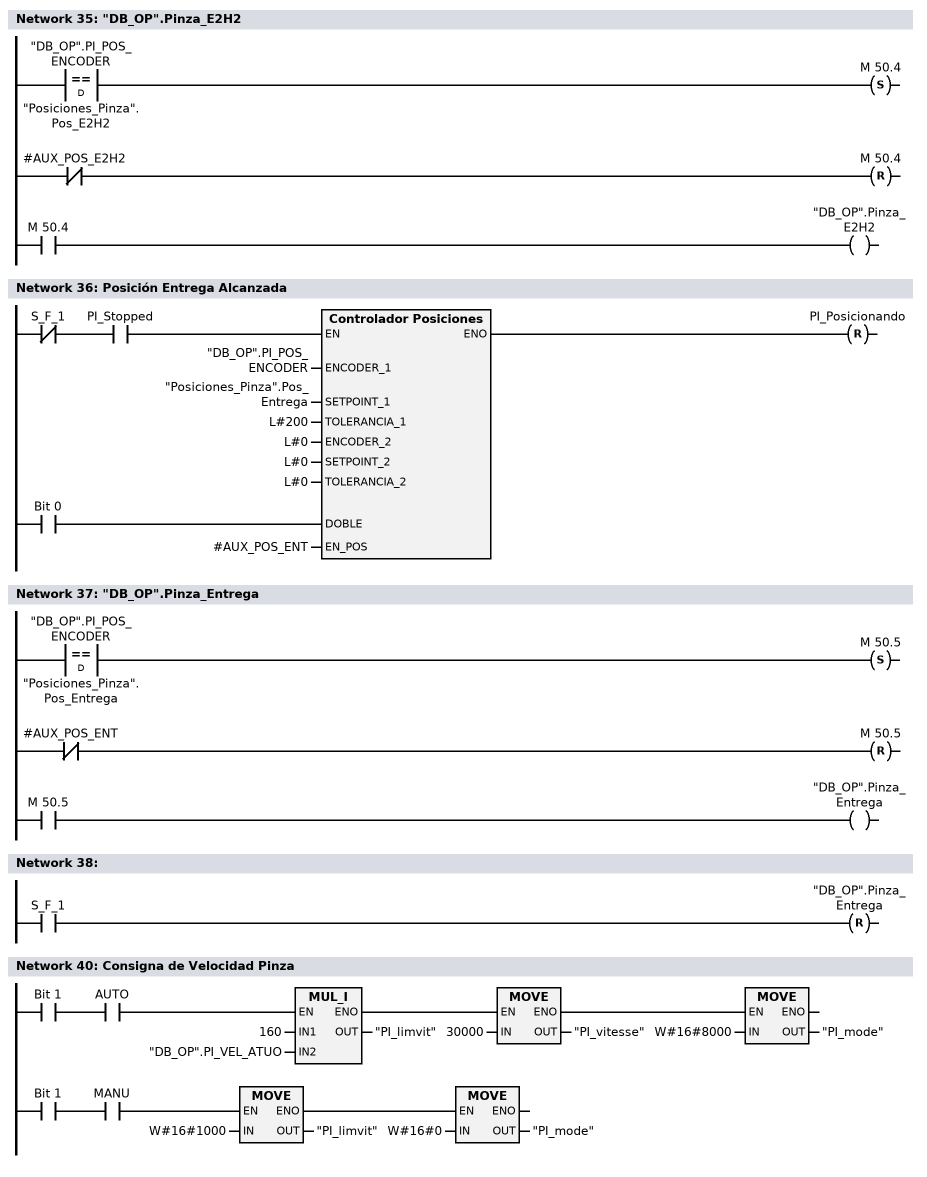
NETWORK
TITLE = "DB_OP".Pinza_E2H2
      A(;
      L     "DB_OP".PI_POS_ENCODER;
      L     "Posiciones_Pinza".Pos_E2H2;
      ==D;
      );
      S     M 50.4;
      AN    #AUX_POS_E2H2;
      R     M 50.4;
      A     M 50.4;
      =     "DB_OP".Pinza_E2H2;
NETWORK
TITLE = Posición Entrega Alcanzada
      A     "Bit 0";
      =     L 85.0;
      BLD   103;
      AN    "S_F_1";
      A     "PI_Stopped";
      JNB   _00b;
      CALL  "Controlador Posiciones" (
           ENCODER_1                := "DB_OP".PI_POS_ENCODER,
           SETPOINT_1               := "Posiciones_Pinza".Pos_Entrega,
           TOLERANCIA_1             := L#200,
           ENCODER_2                := L#0,
           SETPOINT_2               := L#0,
           TOLERANCIA_2             := L#0,
           DOBLE                    := L 85.0,
           EN_POS                   := #AUX_POS_ENT);
_00b: A     BR;
      R     "PI_Posicionando";
NETWORK
TITLE = "DB_OP".Pinza_Entrega
      A(;
      L     "DB_OP".PI_POS_ENCODER;
      L     "Posiciones_Pinza".Pos_Entrega;
      ==D;
      );
      S     M 50.5;
      AN    #AUX_POS_ENT;
      R     M 50.5;
      A     M 50.5;
      =     "DB_OP".Pinza_Entrega;
NETWORK
TITLE =
      A     "S_F_1";
      R     "DB_OP".Pinza_Entrega;
NETWORK
TITLE = ------------ CONSIGNAS DE VELOCIDAD -----------
NETWORK
TITLE = Consigna de Velocidad Pinza
      A     "Bit 1";
      =     L 85.0;
      A(;
      A(;
      A     L 85.0;
      A     "AUTO";
      JNB   _00c;
      L     160;
      L     "DB_OP".PI_VEL_ATUO;
      *I;
      T     "PI_limvit";
      AN    OV;
      SAVE;
      CLR;
_00c: A     BR;
      );
      JNB   _00d;
      L     30000;
      T     "PI_vitesse";
      SET;
      SAVE;
      CLR;
_00d: A     BR;
      );
      JNB   _00e;
      L     W#16#8000;
      T     "PI_mode";
_00e: NOP   0;
      A(;
      A     L 85.0;
      A     "MANU";
      JNB   _00f;
      L     W#16#1000;
      T     "PI_limvit";
      SET;
      SAVE;
      CLR;
_00f: A     BR;
      );
      JNB   _010;
      L     W#16#0;
      T     "PI_mode";
_010: NOP   0;
NETWORK
TITLE = ---------- CÁLCULO DE REFERENCIAS -------------
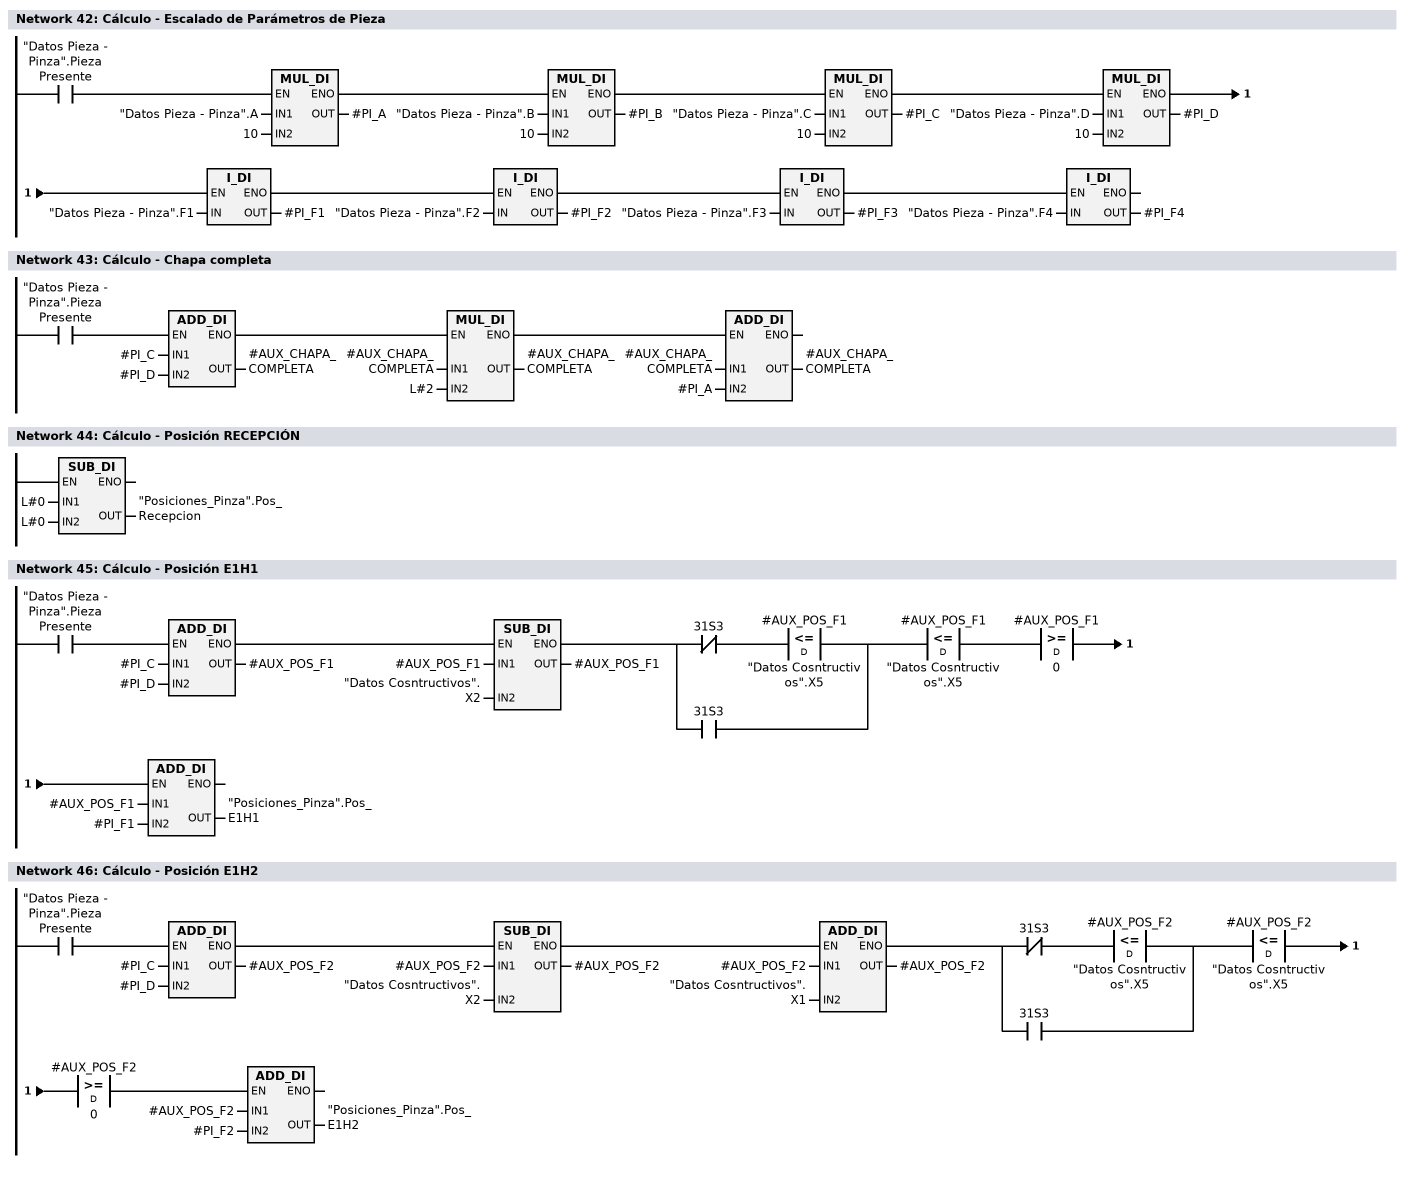
NETWORK
TITLE = Cálculo - Escalado de Parámetros de Pieza 
      A(;
      A(;
      A(;
      A(;
      A(;
      A(;
      A(;
      A     "Datos Pieza - Pinza".PiezaPresente;
      JNB   _011;
      L     "Datos Pieza - Pinza".A;
      L     10;
      *D;
      T     #PI_A;
      AN    OV;
      SAVE;
      CLR;
_011: A     BR;
      );
      JNB   _012;
      L     "Datos Pieza - Pinza".B;
      L     10;
      *D;
      T     #PI_B;
      AN    OV;
      SAVE;
      CLR;
_012: A     BR;
      );
      JNB   _013;
      L     "Datos Pieza - Pinza".C;
      L     10;
      *D;
      T     #PI_C;
      AN    OV;
      SAVE;
      CLR;
_013: A     BR;
      );
      JNB   _014;
      L     "Datos Pieza - Pinza".D;
      L     10;
      *D;
      T     #PI_D;
      AN    OV;
      SAVE;
      CLR;
_014: A     BR;
      );
      JNB   _015;
      L     "Datos Pieza - Pinza".F1;
      ITD;
      T     #PI_F1;
      SET;
      SAVE;
      CLR;
_015: A     BR;
      );
      JNB   _016;
      L     "Datos Pieza - Pinza".F2;
      ITD;
      T     #PI_F2;
      SET;
      SAVE;
      CLR;
_016: A     BR;
      );
      JNB   _017;
      L     "Datos Pieza - Pinza".F3;
      ITD;
      T     #PI_F3;
      SET;
      SAVE;
      CLR;
_017: A     BR;
      );
      JNB   _018;
      L     "Datos Pieza - Pinza".F4;
      ITD;
      T     #PI_F4;
_018: NOP   0;
NETWORK
TITLE = Cálculo - Chapa completa 
      A(;
      A(;
      A     "Datos Pieza - Pinza".PiezaPresente;
      JNB   _019;
      L     #PI_C;
      L     #PI_D;
      +D;
      T     #AUX_CHAPA_COMPLETA;
      AN    OV;
      SAVE;
      CLR;
_019: A     BR;
      );
      JNB   _01a;
      L     #AUX_CHAPA_COMPLETA;
      L     L#2;
      *D;
      T     #AUX_CHAPA_COMPLETA;
      AN    OV;
      SAVE;
      CLR;
_01a: A     BR;
      );
      JNB   _01b;
      L     #AUX_CHAPA_COMPLETA;
      L     #PI_A;
      +D;
      T     #AUX_CHAPA_COMPLETA;
_01b: NOP   0;
NETWORK
TITLE = Cálculo - Posición RECEPCIÓN
      L     L#0;
      L     L#0;
      -D;
      T     "Posiciones_Pinza".Pos_Recepcion;
      NOP   0;
NETWORK
TITLE = Cálculo - Posición E1H1
      A(;
      A(;
      A     "Datos Pieza - Pinza".PiezaPresente;
      JNB   _01c;
      L     #PI_C;
      L     #PI_D;
      +D;
      T     #AUX_POS_F1;
      AN    OV;
      SAVE;
      CLR;
_01c: A     BR;
      );
      JNB   _01d;
      L     #AUX_POS_F1;
      L     "Datos Cosntructivos".X2;
      -D;
      T     #AUX_POS_F1;
      AN    OV;
      SAVE;
      CLR;
_01d: A     BR;
      );
      A(;
      AN    "31S3";
      A(;
      L     #AUX_POS_F1;
      L     "Datos Cosntructivos".X5;
      <=D;
      );
      O     "31S3";
      );
      A(;
      L     #AUX_POS_F1;
      L     "Datos Cosntructivos".X5;
      <=D;
      );
      A(;
      L     #AUX_POS_F1;
      L     0;
      >=D;
      );
      JNB   _01e;
      L     #AUX_POS_F1;
      L     #PI_F1;
      +D;
      T     "Posiciones_Pinza".Pos_E1H1;
_01e: NOP   0;
NETWORK
TITLE = Cálculo - Posición E1H2
      A(;
      A(;
      A(;
      A     "Datos Pieza - Pinza".PiezaPresente;
      JNB   _01f;
      L     #PI_C;
      L     #PI_D;
      +D;
      T     #AUX_POS_F2;
      AN    OV;
      SAVE;
      CLR;
_01f: A     BR;
      );
      JNB   _020;
      L     #AUX_POS_F2;
      L     "Datos Cosntructivos".X2;
      -D;
      T     #AUX_POS_F2;
      AN    OV;
      SAVE;
      CLR;
_020: A     BR;
      );
      JNB   _021;
      L     #AUX_POS_F2;
      L     "Datos Cosntructivos".X1;
      +D;
      T     #AUX_POS_F2;
      AN    OV;
      SAVE;
      CLR;
_021: A     BR;
      );
      A(;
      AN    "31S3";
      A(;
      L     #AUX_POS_F2;
      L     "Datos Cosntructivos".X5;
      <=D;
      );
      O     "31S3";
      );
      A(;
      L     #AUX_POS_F2;
      L     "Datos Cosntructivos".X5;
      <=D;
      );
      A(;
      L     #AUX_POS_F2;
      L     0;
      >=D;
      );
      JNB   _022;
      L     #AUX_POS_F2;
      L     #PI_F2;
      +D;
      T     "Posiciones_Pinza".Pos_E1H2;
_022: NOP   0;
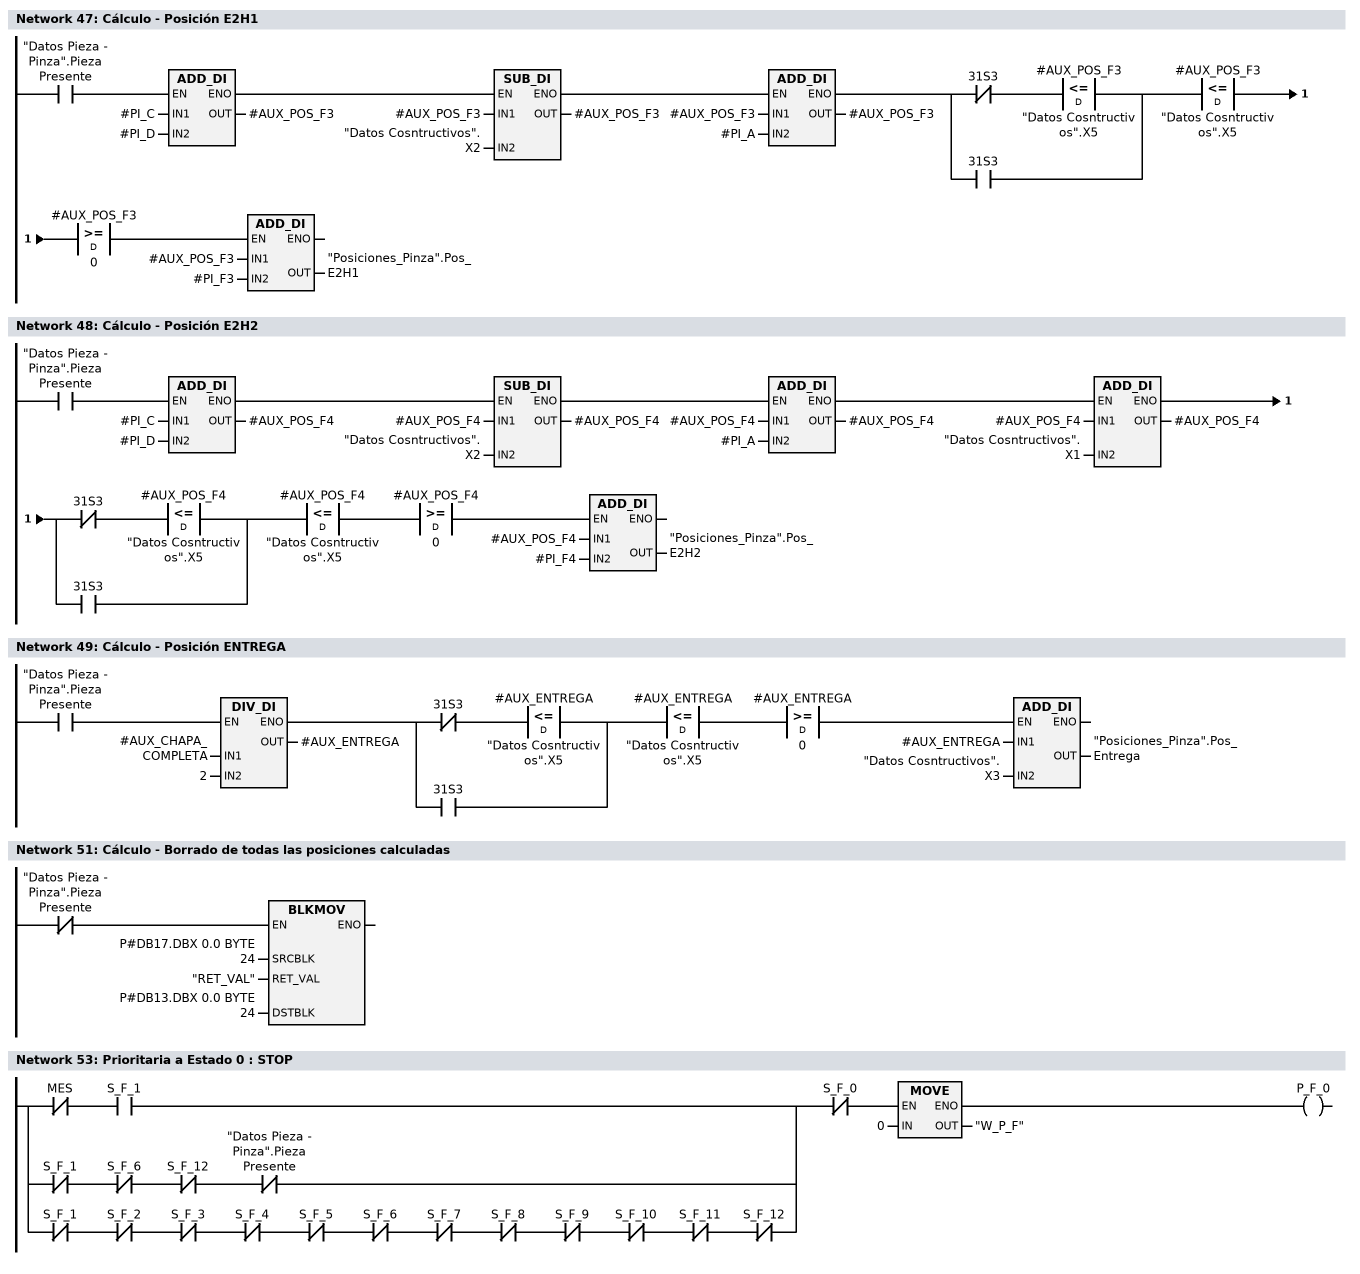
NETWORK
TITLE = Cálculo - Posición E2H1
      A(;
      A(;
      A(;
      A     "Datos Pieza - Pinza".PiezaPresente;
      JNB   _023;
      L     #PI_C;
      L     #PI_D;
      +D;
      T     #AUX_POS_F3;
      AN    OV;
      SAVE;
      CLR;
_023: A     BR;
      );
      JNB   _024;
      L     #AUX_POS_F3;
      L     "Datos Cosntructivos".X2;
      -D;
      T     #AUX_POS_F3;
      AN    OV;
      SAVE;
      CLR;
_024: A     BR;
      );
      JNB   _025;
      L     #AUX_POS_F3;
      L     #PI_A;
      +D;
      T     #AUX_POS_F3;
      AN    OV;
      SAVE;
      CLR;
_025: A     BR;
      );
      A(;
      AN    "31S3";
      A(;
      L     #AUX_POS_F3;
      L     "Datos Cosntructivos".X5;
      <=D;
      );
      O     "31S3";
      );
      A(;
      L     #AUX_POS_F3;
      L     "Datos Cosntructivos".X5;
      <=D;
      );
      A(;
      L     #AUX_POS_F3;
      L     0;
      >=D;
      );
      JNB   _026;
      L     #AUX_POS_F3;
      L     #PI_F3;
      +D;
      T     "Posiciones_Pinza".Pos_E2H1;
_026: NOP   0;
NETWORK
TITLE = Cálculo - Posición E2H2
      A(;
      A(;
      A(;
      A(;
      A     "Datos Pieza - Pinza".PiezaPresente;
      JNB   _027;
      L     #PI_C;
      L     #PI_D;
      +D;
      T     #AUX_POS_F4;
      AN    OV;
      SAVE;
      CLR;
_027: A     BR;
      );
      JNB   _028;
      L     #AUX_POS_F4;
      L     "Datos Cosntructivos".X2;
      -D;
      T     #AUX_POS_F4;
      AN    OV;
      SAVE;
      CLR;
_028: A     BR;
      );
      JNB   _029;
      L     #AUX_POS_F4;
      L     #PI_A;
      +D;
      T     #AUX_POS_F4;
      AN    OV;
      SAVE;
      CLR;
_029: A     BR;
      );
      JNB   _02a;
      L     #AUX_POS_F4;
      L     "Datos Cosntructivos".X1;
      +D;
      T     #AUX_POS_F4;
      AN    OV;
      SAVE;
      CLR;
_02a: A     BR;
      );
      A(;
      AN    "31S3";
      A(;
      L     #AUX_POS_F4;
      L     "Datos Cosntructivos".X5;
      <=D;
      );
      O     "31S3";
      );
      A(;
      L     #AUX_POS_F4;
      L     "Datos Cosntructivos".X5;
      <=D;
      );
      A(;
      L     #AUX_POS_F4;
      L     0;
      >=D;
      );
      JNB   _02b;
      L     #AUX_POS_F4;
      L     #PI_F4;
      +D;
      T     "Posiciones_Pinza".Pos_E2H2;
_02b: NOP   0;
NETWORK
TITLE = Cálculo - Posición ENTREGA
      A(;
      A     "Datos Pieza - Pinza".PiezaPresente;
      JNB   _02c;
      L     #AUX_CHAPA_COMPLETA;
      L     2;
      /D;
      T     #AUX_ENTREGA;
      AN    OV;
      SAVE;
      CLR;
_02c: A     BR;
      );
      A(;
      AN    "31S3";
      A(;
      L     #AUX_ENTREGA;
      L     "Datos Cosntructivos".X5;
      <=D;
      );
      O     "31S3";
      );
      A(;
      L     #AUX_ENTREGA;
      L     "Datos Cosntructivos".X5;
      <=D;
      );
      A(;
      L     #AUX_ENTREGA;
      L     0;
      >=D;
      );
      JNB   _02d;
      L     #AUX_ENTREGA;
      L     "Datos Cosntructivos".X3;
      +D;
      T     "Posiciones_Pinza".Pos_Entrega;
_02d: NOP   0;
NETWORK
TITLE = FC18 - "Registro_pos_Pinza"
      UC    "Registro_pos_Pinza";
NETWORK
TITLE = Cálculo - Borrado de todas las posiciones calculadas 
      AN    "Datos Pieza - Pinza".PiezaPresente;
      JNB   _02e;
      CALL  "BLKMOV" (
           SRCBLK                   := P#DB17.DBX 0.0 BYTE 24,
           RET_VAL                  := "RET_VAL",
           DSTBLK                   := P#DB13.DBX 0.0 BYTE 24);
_02e: NOP   0;
NETWORK
TITLE = ---------- CÁLCULO DE TRANSICIONES ------------
NETWORK
TITLE = Prioritaria a Estado 0 : STOP
      A(;
      AN    "MES";
      A     "S_F_1";
      O;
      AN    "S_F_1";
      AN    "S_F_6";
      AN    "S_F_12";
      AN    "Datos Pieza - Pinza".PiezaPresente;
      O;
      AN    "S_F_1";
      AN    "S_F_2";
      AN    "S_F_3";
      AN    "S_F_4";
      AN    "S_F_5";
      AN    "S_F_6";
      AN    "S_F_7";
      AN    "S_F_8";
      AN    "S_F_9";
      AN    "S_F_10";
      AN    "S_F_11";
      AN    "S_F_12";
      );
      AN    "S_F_0";
      JNB   _02f;
      L     0;
      T     "W_P_F";
      SET;
      SAVE;
      CLR;
_02f: A     BR;
      =     "P_F_0";
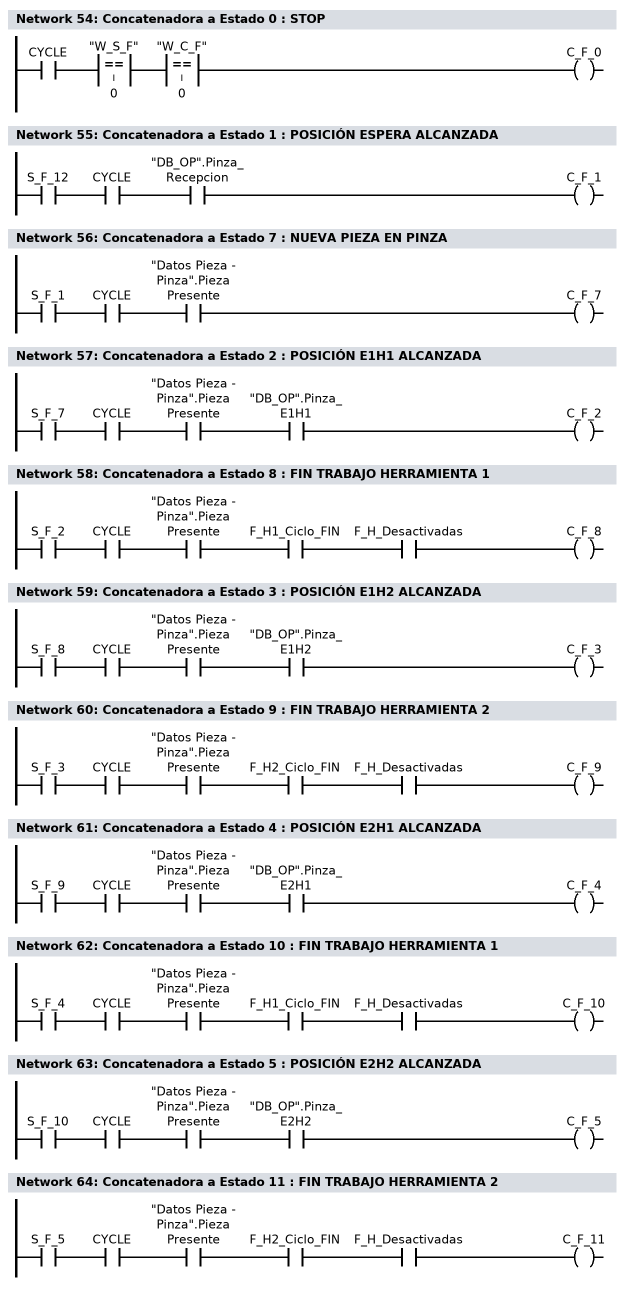
NETWORK
TITLE = Concatenadora a Estado 0 : STOP
      A     "CYCLE";
      A(;
      L     "W_S_F";
      L     0;
      ==I;
      );
      A(;
      L     "W_C_F";
      L     0;
      ==I;
      );
      =     "C_F_0";
NETWORK
TITLE = Concatenadora a Estado 1 : POSICIÓN ESPERA ALCANZADA
      A     "S_F_12";
      A     "CYCLE";
      A     "DB_OP".Pinza_Recepcion;
      =     "C_F_1";
NETWORK
TITLE = Concatenadora a Estado 7 : NUEVA PIEZA EN PINZA
      A     "S_F_1";
      A     "CYCLE";
      A     "Datos Pieza - Pinza".PiezaPresente;
      =     "C_F_7";
NETWORK
TITLE = Concatenadora a Estado 2 : POSICIÓN E1H1 ALCANZADA
      A     "S_F_7";
      A     "CYCLE";
      A     "Datos Pieza - Pinza".PiezaPresente;
      A     "DB_OP".Pinza_E1H1;
      =     "C_F_2";
NETWORK
TITLE = Concatenadora a Estado 8 : FIN TRABAJO HERRAMIENTA 1
      A     "S_F_2";
      A     "CYCLE";
      A     "Datos Pieza - Pinza".PiezaPresente;
      A     "F_H1_Ciclo_FIN";
      A     "F_H_Desactivadas";
      =     "C_F_8";
NETWORK
TITLE = Concatenadora a Estado 3 : POSICIÓN E1H2 ALCANZADA
      A     "S_F_8";
      A     "CYCLE";
      A     "Datos Pieza - Pinza".PiezaPresente;
      A     "DB_OP".Pinza_E1H2;
      =     "C_F_3";
NETWORK
TITLE = Concatenadora a Estado 9 : FIN TRABAJO HERRAMIENTA 2
      A     "S_F_3";
      A     "CYCLE";
      A     "Datos Pieza - Pinza".PiezaPresente;
      A     "F_H2_Ciclo_FIN";
      A     "F_H_Desactivadas";
      =     "C_F_9";
NETWORK
TITLE = Concatenadora a Estado 4 : POSICIÓN E2H1 ALCANZADA
      A     "S_F_9";
      A     "CYCLE";
      A     "Datos Pieza - Pinza".PiezaPresente;
      A     "DB_OP".Pinza_E2H1;
      =     "C_F_4";
NETWORK
TITLE = Concatenadora a Estado 10 : FIN TRABAJO HERRAMIENTA 1
      A     "S_F_4";
      A     "CYCLE";
      A     "Datos Pieza - Pinza".PiezaPresente;
      A     "F_H1_Ciclo_FIN";
      A     "F_H_Desactivadas";
      =     "C_F_10";
NETWORK
TITLE = Concatenadora a Estado 5 : POSICIÓN E2H2 ALCANZADA
      A     "S_F_10";
      A     "CYCLE";
      A     "Datos Pieza - Pinza".PiezaPresente;
      A     "DB_OP".Pinza_E2H2;
      =     "C_F_5";
NETWORK
TITLE = Concatenadora a Estado 11 : FIN TRABAJO HERRAMIENTA 2
      A     "S_F_5";
      A     "CYCLE";
      A     "Datos Pieza - Pinza".PiezaPresente;
      A     "F_H2_Ciclo_FIN";
      A     "F_H_Desactivadas";
      =     "C_F_11";
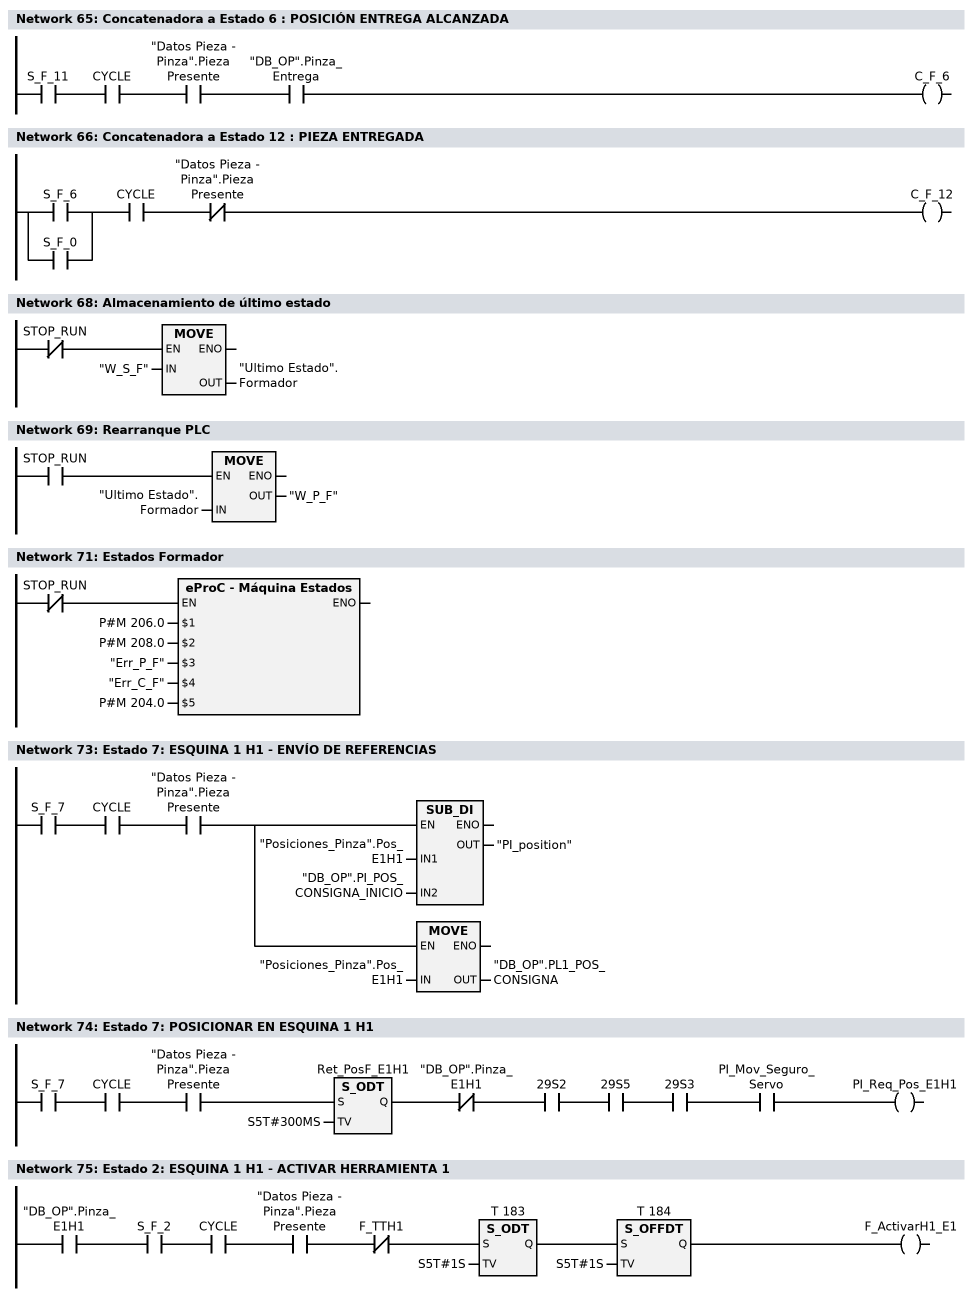
NETWORK
TITLE = Concatenadora a Estado 6 : POSICIÓN ENTREGA ALCANZADA
      A     "S_F_11";
      A     "CYCLE";
      A     "Datos Pieza - Pinza".PiezaPresente;
      A     "DB_OP".Pinza_Entrega;
      =     "C_F_6";
NETWORK
TITLE = Concatenadora a Estado 12 : PIEZA ENTREGADA
      A(;
      O     "S_F_6";
      O     "S_F_0";
      );
      A     "CYCLE";
      AN    "Datos Pieza - Pinza".PiezaPresente;
      =     "C_F_12";
NETWORK
TITLE = ------------ REARRANQUE DE PLC ----------------
NETWORK
TITLE = Almacenamiento de último estado
      AN    "STOP_RUN";
      JNB   _030;
      L     "W_S_F";
      T     "Ultimo Estado".Formador;
_030: NOP   0;
NETWORK
TITLE = Rearranque PLC
      A     "STOP_RUN";
      JNB   _031;
      L     "Ultimo Estado".Formador;
      T     "W_P_F";
_031: NOP   0;
NETWORK
TITLE = ----------- MÁQUINA DE ESTADOS ----------------
NETWORK
TITLE = Estados Formador
      AN    "STOP_RUN";
      JNB   _032;
      CALL  "eProC - Máquina Estados" (
           $1                       := P#M 206.0,
           $2                       := P#M 208.0,
           $3                       := "Err_P_F",
           $4                       := "Err_C_F",
           $5                       := P#M 204.0);
_032: NOP   0;
NETWORK
TITLE = --------- GENERACIÓN DE INSTRUCCIONES ---------
NETWORK
TITLE = Estado 7: ESQUINA 1 H1 - ENVÍO DE REFERENCIAS
      A     "S_F_7";
      A     "CYCLE";
      A     "Datos Pieza - Pinza".PiezaPresente;
      =     L 85.0;
      A     L 85.0;
      JNB   _033;
      L     "Posiciones_Pinza".Pos_E1H1;
      L     "DB_OP".PI_POS_CONSIGNA_INICIO;
      -D;
      T     "PI_position";
_033: NOP   0;
      A     L 85.0;
      JNB   _034;
      L     "Posiciones_Pinza".Pos_E1H1;
      T     "DB_OP".PL1_POS_CONSIGNA;
_034: NOP   0;
NETWORK
TITLE = Estado 7: POSICIONAR EN ESQUINA 1 H1 
      A(;
      A     "S_F_7";
      A     "CYCLE";
      A     "Datos Pieza - Pinza".PiezaPresente;
      L     S5T#300MS;
      SD    "Ret_PosF_E1H1";
      NOP   0;
      NOP   0;
      NOP   0;
      A     "Ret_PosF_E1H1";
      );
      AN    "DB_OP".Pinza_E1H1;
      A     "29S2";
      A     "29S5";
      A     "29S3";
      A     "PI_Mov_Seguro_Servo";
      =     "PI_Req_Pos_E1H1";
NETWORK
TITLE = Estado 2: ESQUINA 1 H1 - ACTIVAR HERRAMIENTA 1
      A(;
      A     "DB_OP".Pinza_E1H1;
      A     "S_F_2";
      A     "CYCLE";
      A     "Datos Pieza - Pinza".PiezaPresente;
      AN    "F_TTH1";
      L     S5T#1S;
      SD    T 183;
      NOP   0;
      NOP   0;
      NOP   0;
      A     T 183;
      );
      L     S5T#1S;
      SF    T 184;
      NOP   0;
      NOP   0;
      NOP   0;
      A     T 184;
      =     "F_ActivarH1_E1";
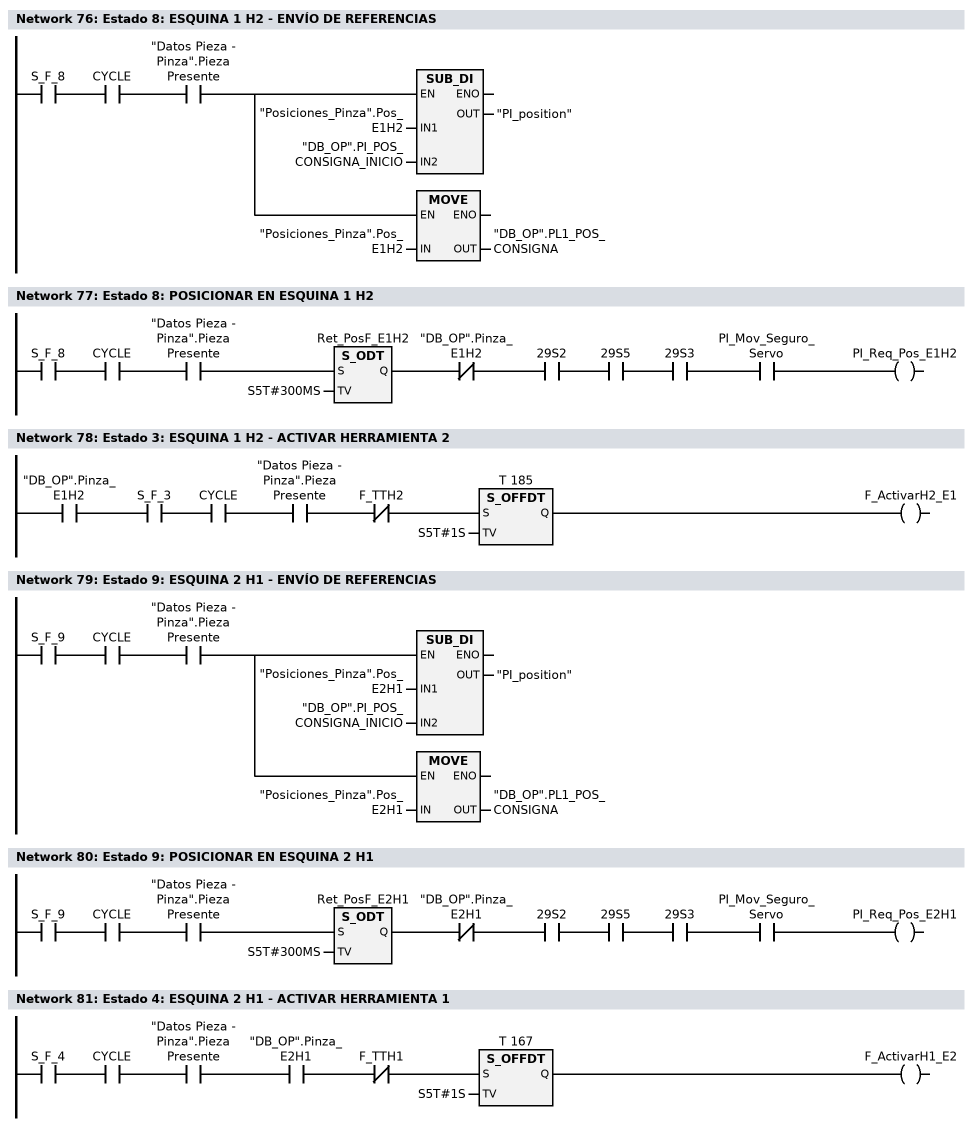
NETWORK
TITLE = Estado 8: ESQUINA 1 H2 - ENVÍO DE REFERENCIAS
      A     "S_F_8";
      A     "CYCLE";
      A     "Datos Pieza - Pinza".PiezaPresente;
      =     L 85.0;
      A     L 85.0;
      JNB   _035;
      L     "Posiciones_Pinza".Pos_E1H2;
      L     "DB_OP".PI_POS_CONSIGNA_INICIO;
      -D;
      T     "PI_position";
_035: NOP   0;
      A     L 85.0;
      JNB   _036;
      L     "Posiciones_Pinza".Pos_E1H2;
      T     "DB_OP".PL1_POS_CONSIGNA;
_036: NOP   0;
NETWORK
TITLE = Estado 8: POSICIONAR EN ESQUINA 1 H2 
      A(;
      A     "S_F_8";
      A     "CYCLE";
      A     "Datos Pieza - Pinza".PiezaPresente;
      L     S5T#300MS;
      SD    "Ret_PosF_E1H2";
      NOP   0;
      NOP   0;
      NOP   0;
      A     "Ret_PosF_E1H2";
      );
      AN    "DB_OP".Pinza_E1H2;
      A     "29S2";
      A     "29S5";
      A     "29S3";
      A     "PI_Mov_Seguro_Servo";
      =     "PI_Req_Pos_E1H2";
NETWORK
TITLE = Estado 3: ESQUINA 1 H2 - ACTIVAR HERRAMIENTA 2
      A     "DB_OP".Pinza_E1H2;
      A     "S_F_3";
      A     "CYCLE";
      A     "Datos Pieza - Pinza".PiezaPresente;
      AN    "F_TTH2";
      L     S5T#1S;
      SF    T 185;
      NOP   0;
      NOP   0;
      NOP   0;
      A     T 185;
      =     "F_ActivarH2_E1";
NETWORK
TITLE = Estado 9: ESQUINA 2 H1 - ENVÍO DE REFERENCIAS
      A     "S_F_9";
      A     "CYCLE";
      A     "Datos Pieza - Pinza".PiezaPresente;
      =     L 85.0;
      A     L 85.0;
      JNB   _037;
      L     "Posiciones_Pinza".Pos_E2H1;
      L     "DB_OP".PI_POS_CONSIGNA_INICIO;
      -D;
      T     "PI_position";
_037: NOP   0;
      A     L 85.0;
      JNB   _038;
      L     "Posiciones_Pinza".Pos_E2H1;
      T     "DB_OP".PL1_POS_CONSIGNA;
_038: NOP   0;
NETWORK
TITLE = Estado 9: POSICIONAR EN ESQUINA 2 H1 
      A(;
      A     "S_F_9";
      A     "CYCLE";
      A     "Datos Pieza - Pinza".PiezaPresente;
      L     S5T#300MS;
      SD    "Ret_PosF_E2H1";
      NOP   0;
      NOP   0;
      NOP   0;
      A     "Ret_PosF_E2H1";
      );
      AN    "DB_OP".Pinza_E2H1;
      A     "29S2";
      A     "29S5";
      A     "29S3";
      A     "PI_Mov_Seguro_Servo";
      =     "PI_Req_Pos_E2H1";
NETWORK
TITLE = Estado 4: ESQUINA 2 H1 - ACTIVAR HERRAMIENTA 1
      A     "S_F_4";
      A     "CYCLE";
      A     "Datos Pieza - Pinza".PiezaPresente;
      A     "DB_OP".Pinza_E2H1;
      AN    "F_TTH1";
      L     S5T#1S;
      SF    T 167;
      NOP   0;
      NOP   0;
      NOP   0;
      A     T 167;
      =     "F_ActivarH1_E2";
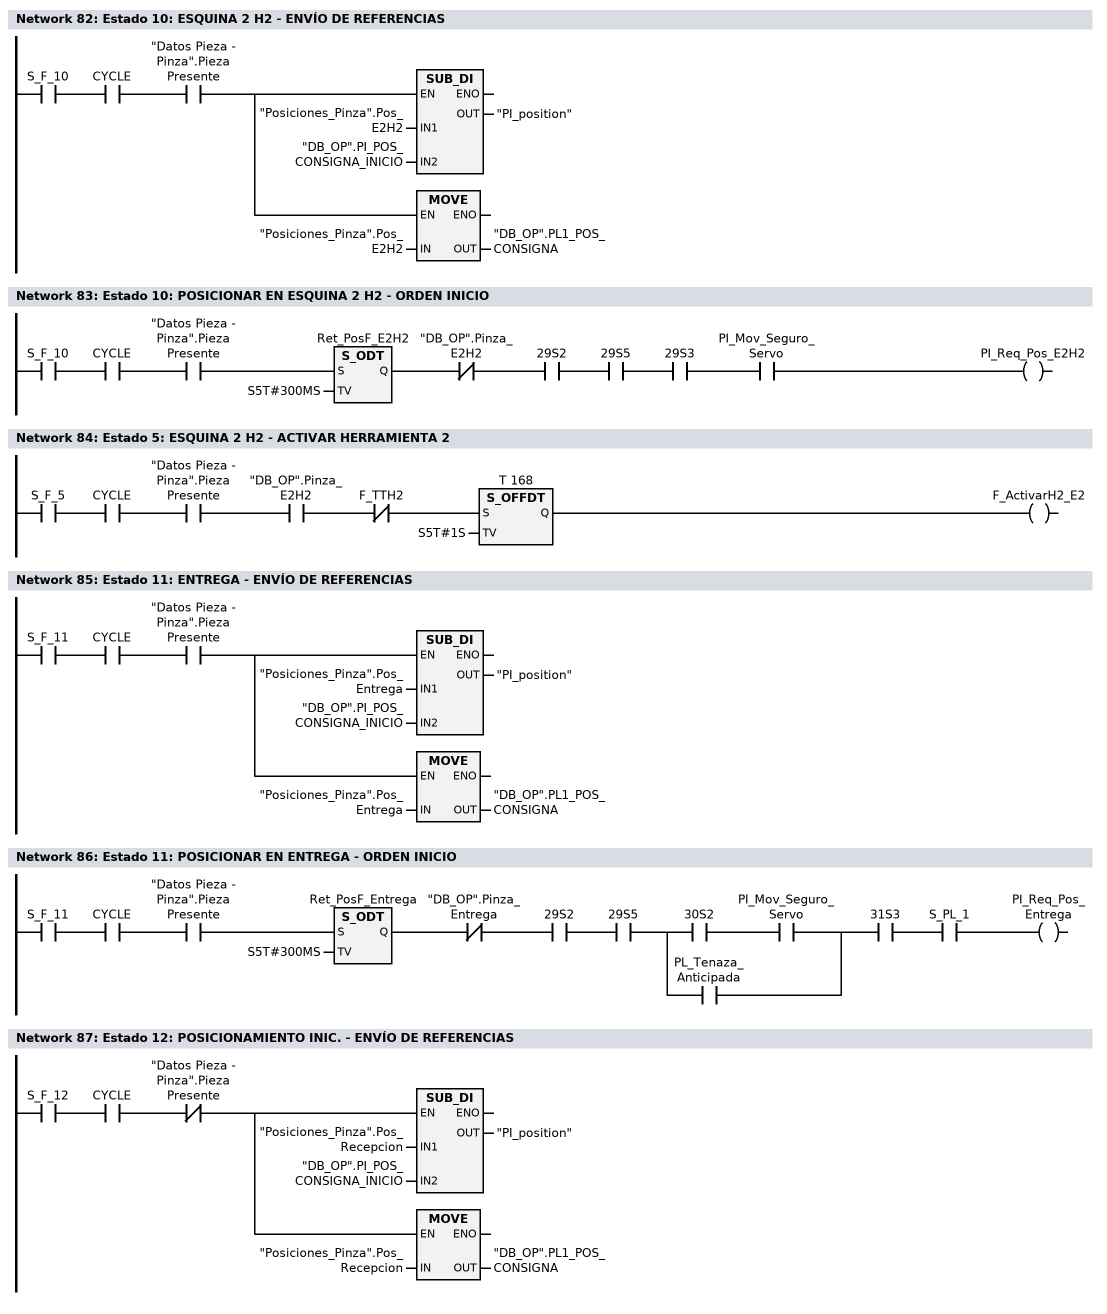
NETWORK
TITLE = Estado 10: ESQUINA 2 H2 - ENVÍO DE REFERENCIAS
      A     "S_F_10";
      A     "CYCLE";
      A     "Datos Pieza - Pinza".PiezaPresente;
      =     L 85.0;
      A     L 85.0;
      JNB   _039;
      L     "Posiciones_Pinza".Pos_E2H2;
      L     "DB_OP".PI_POS_CONSIGNA_INICIO;
      -D;
      T     "PI_position";
_039: NOP   0;
      A     L 85.0;
      JNB   _03a;
      L     "Posiciones_Pinza".Pos_E2H2;
      T     "DB_OP".PL1_POS_CONSIGNA;
_03a: NOP   0;
NETWORK
TITLE = Estado 10: POSICIONAR EN ESQUINA 2 H2 - ORDEN INICIO
      A(;
      A     "S_F_10";
      A     "CYCLE";
      A     "Datos Pieza - Pinza".PiezaPresente;
      L     S5T#300MS;
      SD    "Ret_PosF_E2H2";
      NOP   0;
      NOP   0;
      NOP   0;
      A     "Ret_PosF_E2H2";
      );
      AN    "DB_OP".Pinza_E2H2;
      A     "29S2";
      A     "29S5";
      A     "29S3";
      A     "PI_Mov_Seguro_Servo";
      =     "PI_Req_Pos_E2H2";
NETWORK
TITLE = Estado 5: ESQUINA 2 H2 - ACTIVAR HERRAMIENTA 2
      A     "S_F_5";
      A     "CYCLE";
      A     "Datos Pieza - Pinza".PiezaPresente;
      A     "DB_OP".Pinza_E2H2;
      AN    "F_TTH2";
      L     S5T#1S;
      SF    T 168;
      NOP   0;
      NOP   0;
      NOP   0;
      A     T 168;
      =     "F_ActivarH2_E2";
NETWORK
TITLE = Estado 11: ENTREGA - ENVÍO DE REFERENCIAS
      A     "S_F_11";
      A     "CYCLE";
      A     "Datos Pieza - Pinza".PiezaPresente;
      =     L 85.0;
      A     L 85.0;
      JNB   _03b;
      L     "Posiciones_Pinza".Pos_Entrega;
      L     "DB_OP".PI_POS_CONSIGNA_INICIO;
      -D;
      T     "PI_position";
_03b: NOP   0;
      A     L 85.0;
      JNB   _03c;
      L     "Posiciones_Pinza".Pos_Entrega;
      T     "DB_OP".PL1_POS_CONSIGNA;
_03c: NOP   0;
NETWORK
TITLE = Estado 11: POSICIONAR EN ENTREGA - ORDEN INICIO
      A(;
      A     "S_F_11";
      A     "CYCLE";
      A     "Datos Pieza - Pinza".PiezaPresente;
      L     S5T#300MS;
      SD    "Ret_PosF_Entrega";
      NOP   0;
      NOP   0;
      NOP   0;
      A     "Ret_PosF_Entrega";
      );
      AN    "DB_OP".Pinza_Entrega;
      A     "29S2";
      A     "29S5";
      A(;
      A     "30S2";
      A     "PI_Mov_Seguro_Servo";
      O     "PL_Tenaza_Anticipada";
      );
      A     "31S3";
      A     "S_PL_1";
      =     "PI_Req_Pos_Entrega";
NETWORK
TITLE = Estado 12: POSICIONAMIENTO INIC. - ENVÍO DE REFERENCIAS
      A     "S_F_12";
      A     "CYCLE";
      AN    "Datos Pieza - Pinza".PiezaPresente;
      =     L 85.0;
      A     L 85.0;
      JNB   _03d;
      L     "Posiciones_Pinza".Pos_Recepcion;
      L     "DB_OP".PI_POS_CONSIGNA_INICIO;
      -D;
      T     "PI_position";
_03d: NOP   0;
      A     L 85.0;
      JNB   _03e;
      L     "Posiciones_Pinza".Pos_Recepcion;
      T     "DB_OP".PL1_POS_CONSIGNA;
_03e: NOP   0;
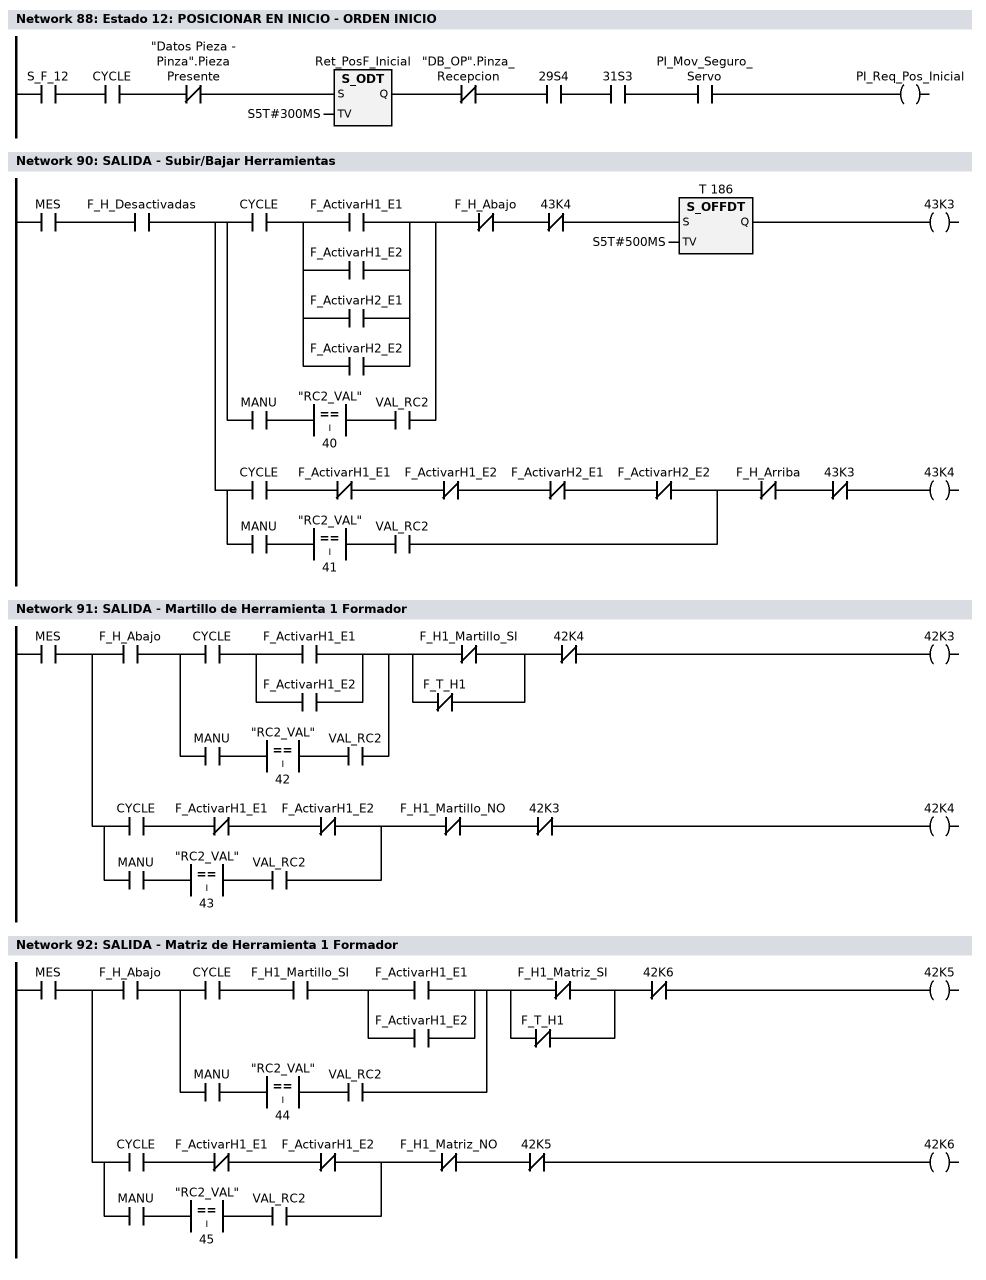
NETWORK
TITLE = Estado 12: POSICIONAR EN INICIO - ORDEN INICIO
      A(;
      A     "S_F_12";
      A     "CYCLE";
      AN    "Datos Pieza - Pinza".PiezaPresente;
      L     S5T#300MS;
      SD    "Ret_PosF_Inicial";
      NOP   0;
      NOP   0;
      NOP   0;
      A     "Ret_PosF_Inicial";
      );
      AN    "DB_OP".Pinza_Recepcion;
      A     "29S4";
      A     "31S3";
      A     "PI_Mov_Seguro_Servo";
      =     "PI_Req_Pos_Inicial";
NETWORK
TITLE = -------------- ACTIVACIÓN DE SALIDAS ----------------
NETWORK
TITLE = SALIDA - Subir/Bajar Herramientas
      A     "MES";
      A     "F_H_Desactivadas";
      =     L 85.0;
      A     L 85.0;
      A(;
      A     "CYCLE";
      A(;
      O     "F_ActivarH1_E1";
      O     "F_ActivarH1_E2";
      O     "F_ActivarH2_E1";
      O     "F_ActivarH2_E2";
      );
      O;
      A     "MANU";
      A(;
      L     "RC2_VAL";
      L     40;
      ==I;
      );
      A     "VAL_RC2";
      );
      AN    "F_H_Abajo";
      AN    "43K4";
      L     S5T#500MS;
      SF    T 186;
      NOP   0;
      NOP   0;
      NOP   0;
      A     T 186;
      =     "43K3";
      A     L 85.0;
      A(;
      A     "CYCLE";
      AN    "F_ActivarH1_E1";
      AN    "F_ActivarH1_E2";
      AN    "F_ActivarH2_E1";
      AN    "F_ActivarH2_E2";
      O;
      A     "MANU";
      A(;
      L     "RC2_VAL";
      L     41;
      ==I;
      );
      A     "VAL_RC2";
      );
      AN    "F_H_Arriba";
      AN    "43K3";
      =     "43K4";
NETWORK
TITLE = SALIDA - Martillo de Herramienta 1 Formador
      A     "MES";
      =     L 85.0;
      A     L 85.0;
      A     "F_H_Abajo";
      A(;
      A     "CYCLE";
      A(;
      O     "F_ActivarH1_E1";
      O     "F_ActivarH1_E2";
      );
      O;
      A     "MANU";
      A(;
      L     "RC2_VAL";
      L     42;
      ==I;
      );
      A     "VAL_RC2";
      );
      A(;
      ON    "F_H1_Martillo_SI";
      ON    "F_T_H1";
      );
      AN    "42K4";
      =     "42K3";
      A     L 85.0;
      A(;
      A     "CYCLE";
      AN    "F_ActivarH1_E1";
      AN    "F_ActivarH1_E2";
      O;
      A     "MANU";
      A(;
      L     "RC2_VAL";
      L     43;
      ==I;
      );
      A     "VAL_RC2";
      );
      AN    "F_H1_Martillo_NO";
      AN    "42K3";
      =     "42K4";
NETWORK
TITLE = SALIDA - Matriz de Herramienta 1 Formador
      A     "MES";
      =     L 85.0;
      A     L 85.0;
      A     "F_H_Abajo";
      A(;
      A     "CYCLE";
      A     "F_H1_Martillo_SI";
      A(;
      O     "F_ActivarH1_E1";
      O     "F_ActivarH1_E2";
      );
      O;
      A     "MANU";
      A(;
      L     "RC2_VAL";
      L     44;
      ==I;
      );
      A     "VAL_RC2";
      );
      A(;
      ON    "F_H1_Matriz_SI";
      ON    "F_T_H1";
      );
      AN    "42K6";
      =     "42K5";
      A     L 85.0;
      A(;
      A     "CYCLE";
      AN    "F_ActivarH1_E1";
      AN    "F_ActivarH1_E2";
      O;
      A     "MANU";
      A(;
      L     "RC2_VAL";
      L     45;
      ==I;
      );
      A     "VAL_RC2";
      );
      AN    "F_H1_Matriz_NO";
      AN    "42K5";
      =     "42K6";
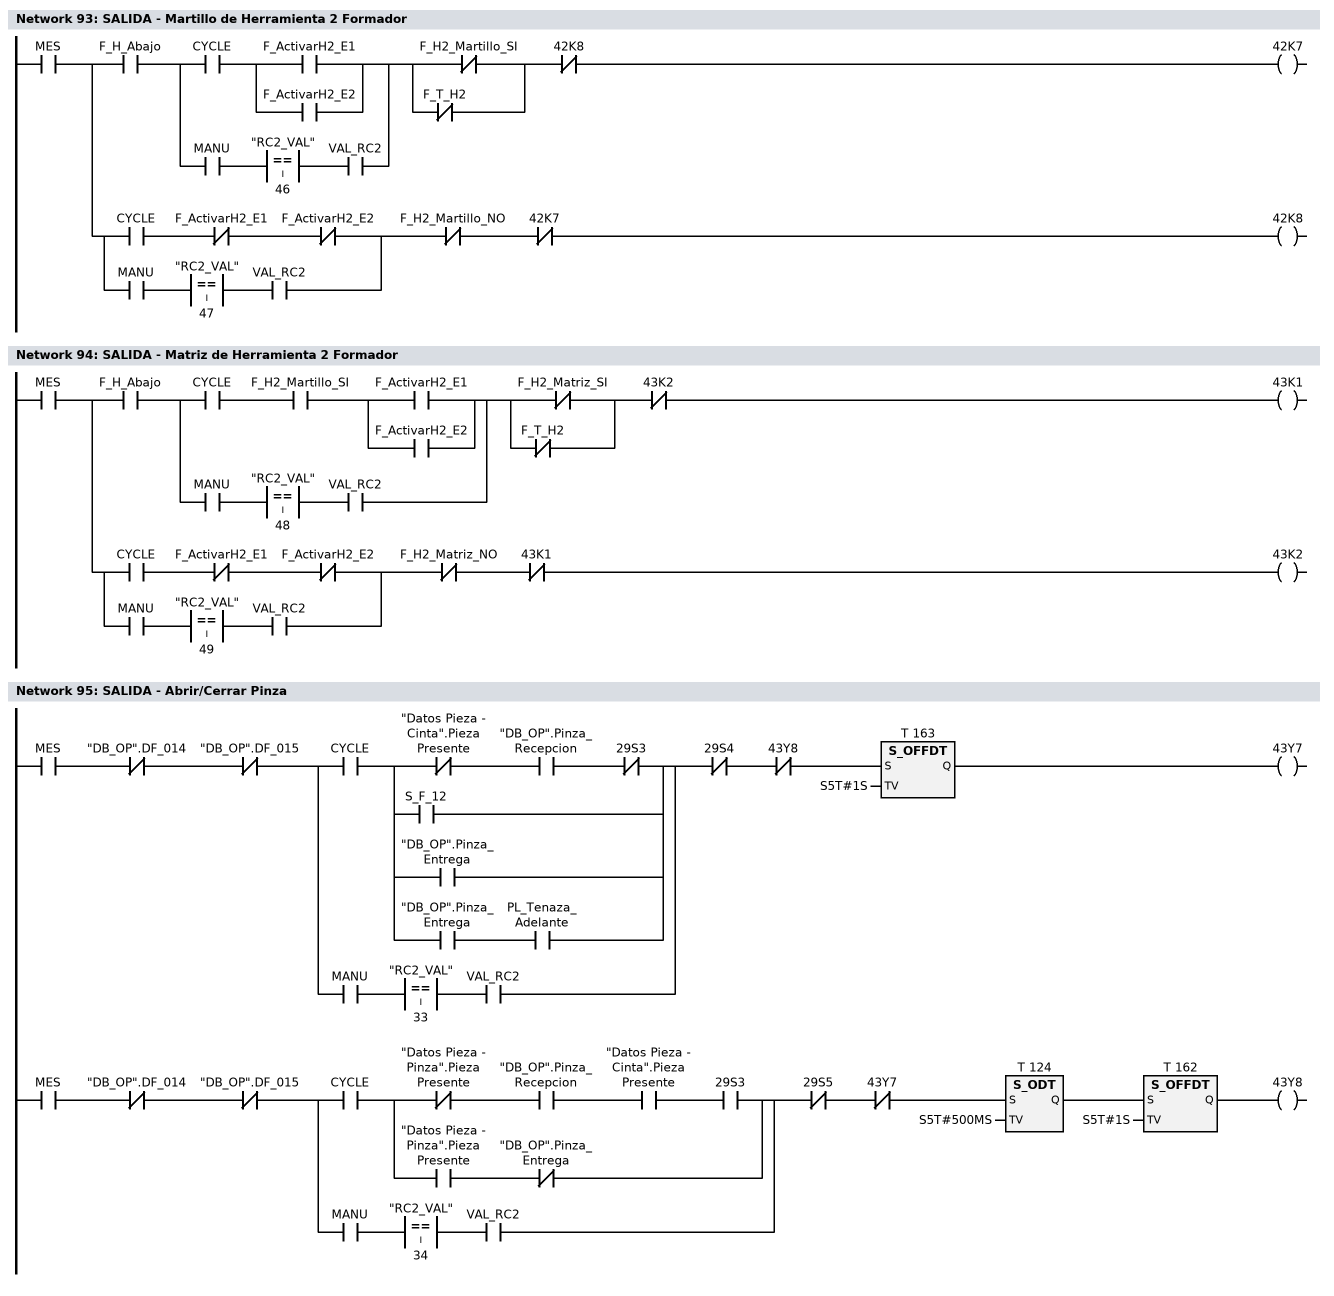
NETWORK
TITLE = SALIDA - Martillo de Herramienta 2 Formador
      A     "MES";
      =     L 85.0;
      A     L 85.0;
      A     "F_H_Abajo";
      A(;
      A     "CYCLE";
      A(;
      O     "F_ActivarH2_E1";
      O     "F_ActivarH2_E2";
      );
      O;
      A     "MANU";
      A(;
      L     "RC2_VAL";
      L     46;
      ==I;
      );
      A     "VAL_RC2";
      );
      A(;
      ON    "F_H2_Martillo_SI";
      ON    "F_T_H2";
      );
      AN    "42K8";
      =     "42K7";
      A     L 85.0;
      A(;
      A     "CYCLE";
      AN    "F_ActivarH2_E1";
      AN    "F_ActivarH2_E2";
      O;
      A     "MANU";
      A(;
      L     "RC2_VAL";
      L     47;
      ==I;
      );
      A     "VAL_RC2";
      );
      AN    "F_H2_Martillo_NO";
      AN    "42K7";
      =     "42K8";
NETWORK
TITLE = SALIDA - Matriz de Herramienta 2 Formador
      A     "MES";
      =     L 85.0;
      A     L 85.0;
      A     "F_H_Abajo";
      A(;
      A     "CYCLE";
      A     "F_H2_Martillo_SI";
      A(;
      O     "F_ActivarH2_E1";
      O     "F_ActivarH2_E2";
      );
      O;
      A     "MANU";
      A(;
      L     "RC2_VAL";
      L     48;
      ==I;
      );
      A     "VAL_RC2";
      );
      A(;
      ON    "F_H2_Matriz_SI";
      ON    "F_T_H2";
      );
      AN    "43K2";
      =     "43K1";
      A     L 85.0;
      A(;
      A     "CYCLE";
      AN    "F_ActivarH2_E1";
      AN    "F_ActivarH2_E2";
      O;
      A     "MANU";
      A(;
      L     "RC2_VAL";
      L     49;
      ==I;
      );
      A     "VAL_RC2";
      );
      AN    "F_H2_Matriz_NO";
      AN    "43K1";
      =     "43K2";
NETWORK
TITLE = SALIDA - Abrir/Cerrar Pinza
      A     "MES";
      AN    "DB_OP".DF_014;
      AN    "DB_OP".DF_015;
      =     L 85.0;
      A     L 85.0;
      A(;
      A     "CYCLE";
      A(;
      AN    "Datos Pieza - Cinta".PiezaPresente;
      A     "DB_OP".Pinza_Recepcion;
      AN    "29S3";
      O     "S_F_12";
      O     "DB_OP".Pinza_Entrega;
      O;
      A     "DB_OP".Pinza_Entrega;
      A     "PL_Tenaza_Adelante";
      );
      O;
      A     "MANU";
      A(;
      L     "RC2_VAL";
      L     33;
      ==I;
      );
      A     "VAL_RC2";
      );
      AN    "29S4";
      AN    "43Y8";
      L     S5T#1S;
      SF    T 163;
      NOP   0;
      NOP   0;
      NOP   0;
      A     T 163;
      =     "43Y7";
      A(;
      A     L 85.0;
      A(;
      A     "CYCLE";
      A(;
      AN    "Datos Pieza - Pinza".PiezaPresente;
      A     "DB_OP".Pinza_Recepcion;
      A     "Datos Pieza - Cinta".PiezaPresente;
      A     "29S3";
      O;
      A     "Datos Pieza - Pinza".PiezaPresente;
      AN    "DB_OP".Pinza_Entrega;
      );
      O;
      A     "MANU";
      A(;
      L     "RC2_VAL";
      L     34;
      ==I;
      );
      A     "VAL_RC2";
      );
      AN    "29S5";
      AN    "43Y7";
      L     S5T#500MS;
      SD    T 124;
      NOP   0;
      NOP   0;
      NOP   0;
      A     T 124;
      );
      L     S5T#1S;
      SF    T 162;
      NOP   0;
      NOP   0;
      NOP   0;
      A     T 162;
      =     "43Y8";
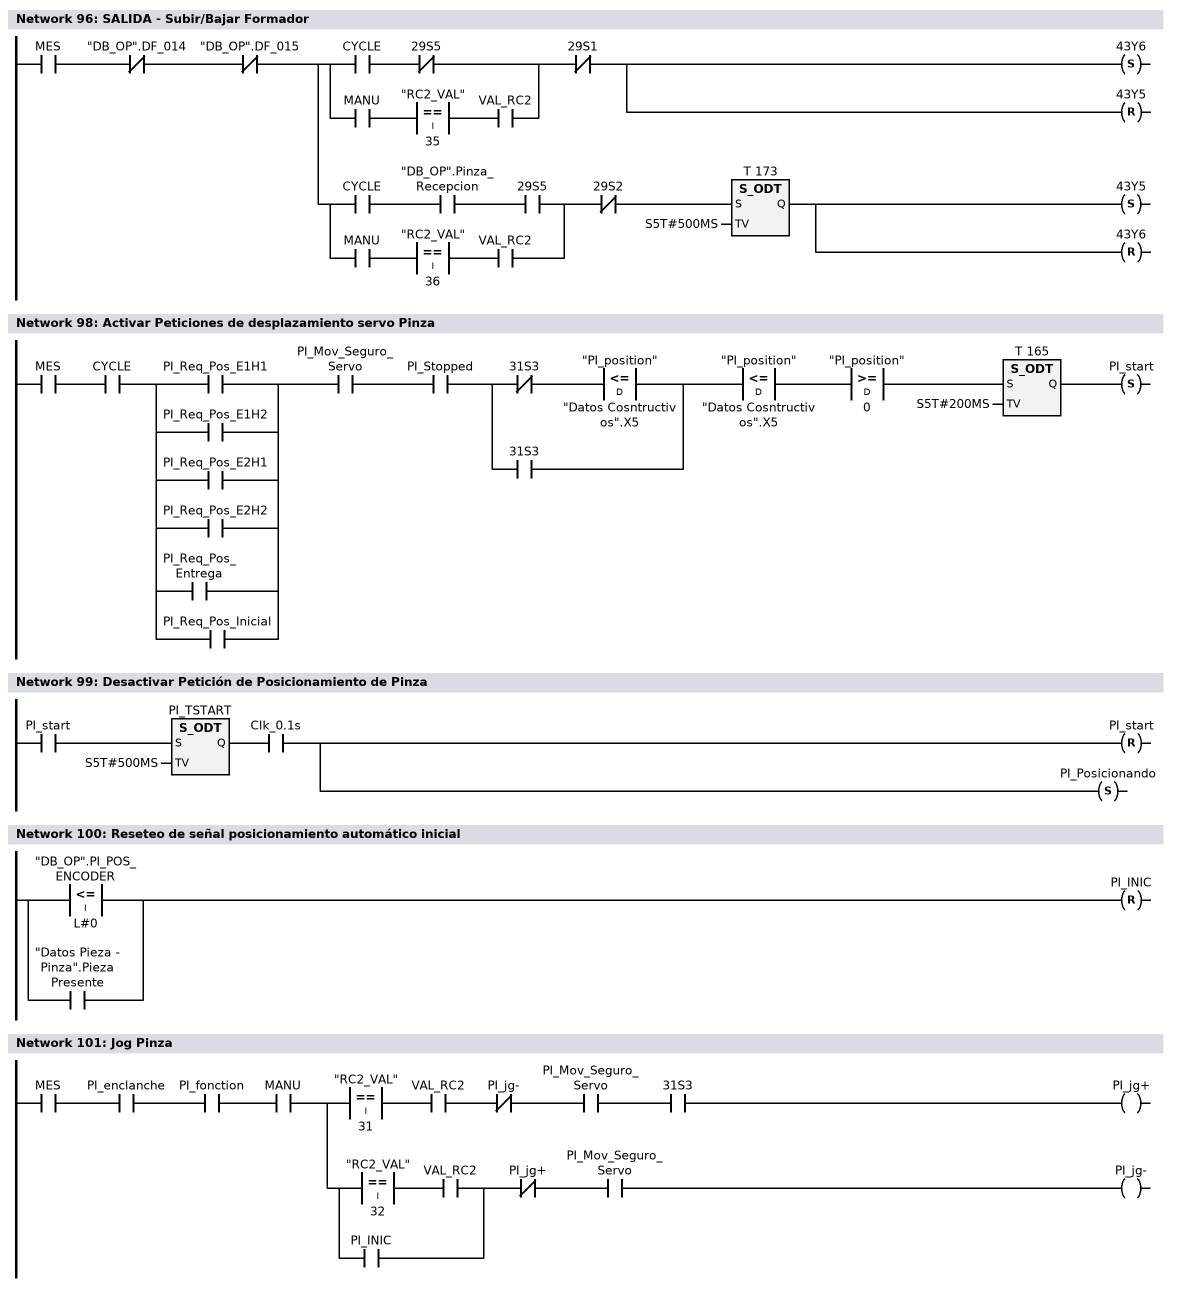
NETWORK
TITLE = SALIDA - Subir/Bajar Formador
      A     "MES";
      AN    "DB_OP".DF_014;
      AN    "DB_OP".DF_015;
      =     L 85.0;
      A     L 85.0;
      A(;
      A     "CYCLE";
      AN    "29S5";
      O;
      A     "MANU";
      A(;
      L     "RC2_VAL";
      L     35;
      ==I;
      );
      A     "VAL_RC2";
      );
      AN    "29S1";
      S     "43Y6";
      R     "43Y5";
      A     L 85.0;
      A(;
      A     "CYCLE";
      A     "DB_OP".Pinza_Recepcion;
      A     "29S5";
      O;
      A     "MANU";
      A(;
      L     "RC2_VAL";
      L     36;
      ==I;
      );
      A     "VAL_RC2";
      );
      AN    "29S2";
      L     S5T#500MS;
      SD    T 173;
      NOP   0;
      NOP   0;
      NOP   0;
      A     T 173;
      S     "43Y5";
      R     "43Y6";
NETWORK
TITLE = -------------- DESPLAZAMIENTO SERVO PINZA ---------------
NETWORK
TITLE = Activar Peticiones de desplazamiento servo Pinza
      A     "MES";
      A     "CYCLE";
      A(;
      O     "PI_Req_Pos_E1H1";
      O     "PI_Req_Pos_E1H2";
      O     "PI_Req_Pos_E2H1";
      O     "PI_Req_Pos_E2H2";
      O     "PI_Req_Pos_Entrega";
      O     "PI_Req_Pos_Inicial";
      );
      A     "PI_Mov_Seguro_Servo";
      A     "PI_Stopped";
      A(;
      AN    "31S3";
      A(;
      L     "PI_position";
      L     "Datos Cosntructivos".X5;
      <=D;
      );
      O     "31S3";
      );
      A(;
      L     "PI_position";
      L     "Datos Cosntructivos".X5;
      <=D;
      );
      A(;
      L     "PI_position";
      L     0;
      >=D;
      );
      L     S5T#200MS;
      SD    T 165;
      NOP   0;
      NOP   0;
      NOP   0;
      A     T 165;
      S     "PI_start";
NETWORK
TITLE = Desactivar Petición de Posicionamiento de Pinza
      A(;
      A     "PI_start";
      L     S5T#500MS;
      SD    "PI_TSTART";
      NOP   0;
      NOP   0;
      NOP   0;
      A     "PI_TSTART";
      );
      A     "Clk_0.1s";
      R     "PI_start";
      S     "PI_Posicionando";
NETWORK
TITLE = Reseteo de señal posicionamiento automático inicial
      O(;
      L     "DB_OP".PI_POS_ENCODER;
      L     L#0;
      <=I;
      );
      O     "Datos Pieza - Pinza".PiezaPresente;
      R     "PI_INIC";
NETWORK
TITLE = Jog Pinza 
      A     "MES";
      A     "PI_enclanche";
      A     "PI_fonction";
      A     "MANU";
      =     L 85.0;
      A     L 85.0;
      A(;
      L     "RC2_VAL";
      L     31;
      ==I;
      );
      A     "VAL_RC2";
      AN    "PI_jg-";
      A     "PI_Mov_Seguro_Servo";
      A     "31S3";
      =     "PI_jg+";
      A     L 85.0;
      A(;
      A(;
      L     "RC2_VAL";
      L     32;
      ==I;
      );
      A     "VAL_RC2";
      O     "PI_INIC";
      );
      AN    "PI_jg+";
      A     "PI_Mov_Seguro_Servo";
      =     "PI_jg-";
NETWORK
TITLE = --------------- CONTROL GRUPO HIDRÁULICO ------------
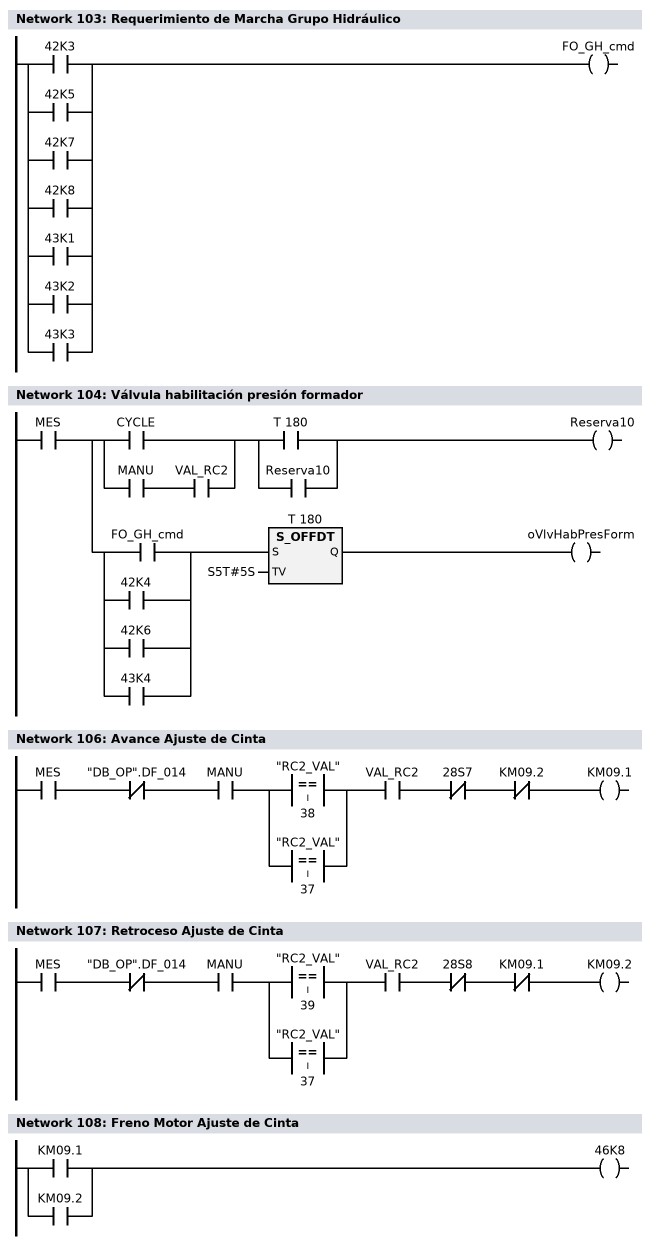
NETWORK
TITLE = Requerimiento de Marcha Grupo Hidráulico 
      O     "42K3";
      O     "42K5";
      O     "42K7";
      O     "42K8";
      O     "43K1";
      O     "43K2";
      O     "43K3";
      =     "FO_GH_cmd";
NETWORK
TITLE = Válvula habilitación presión formador
      A     "MES";
      =     L 85.0;
      A     L 85.0;
      A(;
      O     "CYCLE";
      O;
      A     "MANU";
      A     "VAL_RC2";
      );
      A(;
      O     T 180;
      O     "Reserva10";
      );
      =     "Reserva10";
      A     L 85.0;
      A(;
      O     "FO_GH_cmd";
      O     "42K4";
      O     "42K6";
      O     "43K4";
      );
      L     S5T#5S;
      SF    T 180;
      NOP   0;
      NOP   0;
      NOP   0;
      A     T 180;
      =     "oVlvHabPresForm";
NETWORK
TITLE = ------------ AJUSTE MANUAL ANCHO DE CINTA ----------------
NETWORK
TITLE = Avance Ajuste de Cinta
      A     "MES";
      AN    "DB_OP".DF_014;
      A     "MANU";
      A(;
      O(;
      L     "RC2_VAL";
      L     38;
      ==I;
      );
      O(;
      L     "RC2_VAL";
      L     37;
      ==I;
      );
      );
      A     "VAL_RC2";
      AN    "28S7";
      AN    "KM09.2";
      =     "KM09.1";
NETWORK
TITLE = Retroceso Ajuste de Cinta
      A     "MES";
      AN    "DB_OP".DF_014;
      A     "MANU";
      A(;
      O(;
      L     "RC2_VAL";
      L     39;
      ==I;
      );
      O(;
      L     "RC2_VAL";
      L     37;
      ==I;
      );
      );
      A     "VAL_RC2";
      AN    "28S8";
      AN    "KM09.1";
      =     "KM09.2";
NETWORK
TITLE = Freno Motor Ajuste de Cinta
      O     "KM09.1";
      O     "KM09.2";
      =     "46K8";
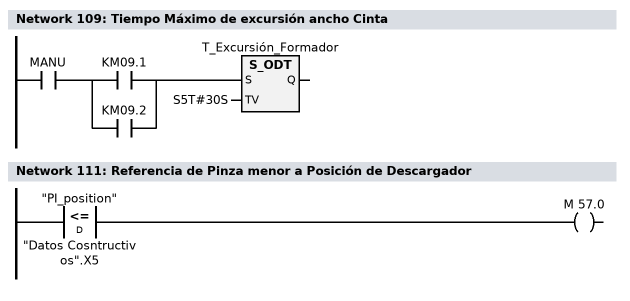
NETWORK
TITLE = Tiempo Máximo de excursión ancho Cinta
      A     "MANU";
      A(;
      O     "KM09.1";
      O     "KM09.2";
      );
      L     S5T#30S;
      SD    "T_Excursión_Formador";
      NOP   0;
      NOP   0;
      NOP   0;
      NOP   0;
NETWORK
TITLE = ------------------------------------------------------------
NETWORK
TITLE = Referencia de Pinza menor a Posición de Descargador
      L     "PI_position";
      L     "Datos Cosntructivos".X5;
      <=D;
      =     M 57.0;
END_FUNCTION

FUNCTION "Controlador Posiciones" : VOID	// FC 13
AUTHOR : EMR
NAME : eProC
VERSION : 0.1
VAR_INPUT
  ENCODER_1 : DINT ;
  SETPOINT_1 : DINT ;
  TOLERANCIA_1 : DINT ;
  ENCODER_2 : DINT ;
  SETPOINT_2 : DINT ;
  TOLERANCIA_2 : DINT ;
  DOBLE : BOOL ;	//Indica si se trabaja con 1 o 2 encóders
END_VAR
VAR_OUTPUT
  EN_POS : BOOL ;
END_VAR
VAR_TEMP
  AUX_INF_2 : DINT ;
  AUX_INF_1 : DINT ;
  AUX_SUP_2 : DINT ;
  AUX_SUP_1 : DINT ;
END_VAR
BEGIN
